LIN {X 0,Y 549.947,Z 550.345,A -85,B 0,C 180,E1 -11066.532,E2 -11066.532} C_VEL
LIN {X 0,Y 549.396,Z 557.599,A -85,B 0,C 180,E1 -11067.808,E2 -11067.808} C_VEL
LIN {X 0,Y 549.182,Z 562.629,A -85,B 0,C 180,E1 -11068.904,E2 -11068.904} C_VEL
LIN {X 0,Y 548.851,Z 567.942,A -85,B 0,C 180,E1 -11070.366,E2 -11070.366} C_VEL
LIN {X 0,Y 548.664,Z 570.891,A -85,B 0,C 180,E1 -11071.463,E2 -11071.463} C_VEL
LIN {X 0,Y 548.707,Z 573.631,A -85,B 0,C 180,E1 -11072.927,E2 -11072.927} C_VEL
LIN {X 0,Y 548.574,Z 575.081,A -85,B 0,C 180,E1 -11074.394,E2 -11074.394} C_VEL
LIN {X 0,Y 548.685,Z 575.22,A -85,B 0,C 180,E1 -11075.862,E2 -11075.862} C_VEL
LIN {X 0,Y 548.777,Z 574.076,A -85,B 0,C 180,E1 -11077.333,E2 -11077.333} C_VEL
LIN {X 0,Y 548.924,Z 571.601,A -85,B 0,C 180,E1 -11078.808,E2 -11078.808} C_VEL
LIN {X 0,Y 549.304,Z 567.682,A -85,B 0,C 180,E1 -11080.284,E2 -11080.284} C_VEL
LIN {X 0,Y 549.668,Z 562.23,A -85,B 0,C 180,E1 -11081.765,E2 -11081.765} C_VEL
LIN {X 0,Y 550.064,Z 557.037,A -85,B 0,C 180,E1 -11082.876,E2 -11082.876} C_VEL
LIN {X 0,Y 550.653,Z 549.525,A -85,B 0,C 180,E1 -11084.174,E2 -11084.174} C_VEL
LIN {X 0,Y 551.216,Z 542.172,A -85,B 0,C 180,E1 -11085.223,E2 -11085.223} C_VEL
LIN {X 0,Y 551.874,Z 532.144,A -85,B 0,C 180,E1 -11086.404,E2 -11086.404} C_VEL
LIN {X 0,Y 552.495,Z 521.544,A -85,B 0,C 180,E1 -11087.429,E2 -11087.429} C_VEL
LIN {X 0,Y 553.106,Z 510.224,A -85,B 0,C 180,E1 -11088.328,E2 -11088.328} C_VEL
LIN {X 0,Y 553.739,Z 498.155,A -85,B 0,C 180,E1 -11089.105,E2 -11089.105} C_VEL
LIN {X 0,Y 554.247,Z 484.443,A -85,B 0,C 180,E1 -11089.807,E2 -11089.807} C_VEL
LIN {X 0,Y 554.553,Z 471.078,A -85,B 0,C 180,E1 -11090.325,E2 -11090.325} C_VEL
LIN {X 0,Y 554.726,Z 456.438,A -85,B 0,C 180,E1 -11090.725,E2 -11090.725} C_VEL
LIN {X 0,Y 554.878,Z 439.3,A -85,B 0,C 180,E1 -11091.001,E2 -11091.001} C_VEL
LIN {X 0,Y 555.689,Z 346.431,A -85,B 0,C 180,E1 -11092.217,E2 -11092.217} C_VEL
LIN {X 0,Y 549.268,Z 330.203,A -85,B 0,C 180,E1 -11092.678,E2 -11092.678} C_VEL
LIN {X 0,Y 549.162,Z 329.646,A -85,B 0,C 180,E1 -11092.721,E2 -11092.721} C_VEL
LIN {X 0,Y 549.175,Z 329.64,A -85,B 0,C 180,E1 -11095.099,E2 -11095.099} C_VEL
LIN {X 0,Y 549.187,Z 329.634,A -85,B 0,C 180,E1 -11098.158,E2 -11098.158} C_VEL
LIN {X 0,Y 549.165,Z 329.637,A -85,B 0,C 180,E1 -11100.677,E2 -11100.677} C_VEL
LIN {X 0,Y 549.119,Z 329.639,A -85,B 0,C 180,E1 -11103.264,E2 -11103.264} C_VEL
LIN {X 0,Y 549.15,Z 329.64,A -85,B 0,C 180,E1 -11105.926,E2 -11105.926} C_VEL
LIN {X 0,Y 549.129,Z 329.638,A -85,B 0,C 180,E1 -11108.914,E2 -11108.914} C_VEL
LIN {X 0,Y 549.137,Z 329.639,A -85,B 0,C 180,E1 -11111.551,E2 -11111.551} C_VEL
LIN {X 0,Y 549.203,Z 329.629,A -85,B 0,C 180,E1 -11114.545,E2 -11114.545} C_VEL
LIN {X 0,Y 549.154,Z 329.636,A -85,B 0,C 180,E1 -11117.467,E2 -11117.467} C_VEL
LIN {X 0,Y 549.137,Z 329.636,A -85,B 0,C 180,E1 -11120.374,E2 -11120.374} C_VEL
LIN {X 0,Y 549.139,Z 329.617,A -85,B 0,C 180,E1 -11123.474,E2 -11123.474} C_VEL
LIN {X 0,Y 549.147,Z 329.637,A -85,B 0,C 180,E1 -11126.005,E2 -11126.005} C_VEL
LIN {X 0,Y 549.161,Z 329.628,A -85,B 0,C 180,E1 -11128.713,E2 -11128.713} C_VEL
LIN {X 0,Y 549.175,Z 329.629,A -85,B 0,C 180,E1 -11131.009,E2 -11131.009} C_VEL
LIN {X 0,Y 549.178,Z 329.634,A -85,B 0,C 180,E1 -11133.486,E2 -11133.486} C_VEL
LIN {X 0,Y 549.163,Z 329.639,A -85,B 0,C 180,E1 -11135.911,E2 -11135.911} C_VEL
LIN {X 0,Y 549.18,Z 329.627,A -85,B 0,C 180,E1 -11139.076,E2 -11139.076} C_VEL
LIN {X 0,Y 549.182,Z 329.642,A -85,B 0,C 180,E1 -11141.406,E2 -11141.406} C_VEL
LIN {X 0,Y 549.194,Z 329.638,A -85,B 0,C 180,E1 -11142.268,E2 -11142.268} C_VEL
LIN {X 0,Y 553.527,Z 343.362,A -85,B 0,C 180,E1 -11142.596,E2 -11142.596} C_VEL
LIN {X 0,Y 552.255,Z 449.713,A -85,B 0,C 180,E1 -11144.222,E2 -11144.222} C_VEL
LIN {X 0,Y 552.112,Z 464.877,A -85,B 0,C 180,E1 -11144.612,E2 -11144.612} C_VEL
LIN {X 0,Y 551.849,Z 479.41,A -85,B 0,C 180,E1 -11145.143,E2 -11145.143} C_VEL
LIN {X 0,Y 551.501,Z 492.173,A -85,B 0,C 180,E1 -11145.754,E2 -11145.754} C_VEL
LIN {X 0,Y 551.121,Z 504.477,A -85,B 0,C 180,E1 -11146.494,E2 -11146.494} C_VEL
LIN {X 0,Y 550.667,Z 516.942,A -85,B 0,C 180,E1 -11147.418,E2 -11147.418} C_VEL
LIN {X 0,Y 550.22,Z 527.741,A -85,B 0,C 180,E1 -11148.39,E2 -11148.39} C_VEL
LIN {X 0,Y 549.971,Z 536.697,A -85,B 0,C 180,E1 -11149.358,E2 -11149.358} C_VEL
LIN {X 0,Y 549.516,Z 545.315,A -85,B 0,C 180,E1 -11150.462,E2 -11150.462} C_VEL
LIN {X 0,Y 549.197,Z 553.545,A -85,B 0,C 180,E1 -11151.75,E2 -11151.75} C_VEL
LIN {X 0,Y 548.936,Z 560.126,A -85,B 0,C 180,E1 -11153.037,E2 -11153.037} C_VEL
LIN {X 0,Y 548.769,Z 564.687,A -85,B 0,C 180,E1 -11154.139,E2 -11154.139} C_VEL
LIN {X 0,Y 548.596,Z 569.27,A -85,B 0,C 180,E1 -11155.606,E2 -11155.606} C_VEL
LIN {X 0,Y 548.655,Z 572.352,A -85,B 0,C 180,E1 -11157.073,E2 -11157.073} C_VEL
LIN {X 0,Y 548.562,Z 574.044,A -85,B 0,C 180,E1 -11158.536,E2 -11158.536} C_VEL
LIN {X 0,Y 548.463,Z 574.349,A -85,B 0,C 180,E1 -11160,E2 -11160} C_VEL
LIN {X 0,Y 548.586,Z 573.208,A -85,B 0,C 180,E1 -11161.463,E2 -11161.463} C_VEL
LIN {X 0,Y 548.967,Z 570.638,A -85,B 0,C 180,E1 -11162.925,E2 -11162.925} C_VEL
LIN {X 0,Y 549.423,Z 566.6,A -85,B 0,C 180,E1 -11164.387,E2 -11164.387} C_VEL
LIN {X 0,Y 549.419,Z 562.553,A -85,B 0,C 180,E1 -11165.487,E2 -11165.487} C_VEL
LIN {X 0,Y 549.926,Z 557.46,A -85,B 0,C 180,E1 -11166.582,E2 -11166.582} C_VEL
LIN {X 0,Y 550.477,Z 550.127,A -85,B 0,C 180,E1 -11167.862,E2 -11167.862} C_VEL
LIN {X 0,Y 550.884,Z 542.443,A -85,B 0,C 180,E1 -11168.961,E2 -11168.961} C_VEL
LIN {X 0,Y 551.383,Z 533.157,A -85,B 0,C 180,E1 -11170.059,E2 -11170.059} C_VEL
LIN {X 0,Y 551.887,Z 522.846,A -85,B 0,C 180,E1 -11171.067,E2 -11171.067} C_VEL
LIN {X 0,Y 552.536,Z 511.383,A -85,B 0,C 180,E1 -11171.981,E2 -11171.981} C_VEL
LIN {X 0,Y 553.175,Z 499.168,A -85,B 0,C 180,E1 -11172.772,E2 -11172.772} C_VEL
LIN {X 0,Y 553.575,Z 486.327,A -85,B 0,C 180,E1 -11173.444,E2 -11173.444} C_VEL
LIN {X 0,Y 553.859,Z 472.723,A -85,B 0,C 180,E1 -11173.997,E2 -11173.997} C_VEL
LIN {X 0,Y 554.047,Z 458.452,A -85,B 0,C 180,E1 -11174.412,E2 -11174.412} C_VEL
LIN {X 0,Y 554.314,Z 436.957,A -85,B 0,C 180,E1 -11174.802,E2 -11174.802} C_VEL
LIN {X 0,Y 556.216,Z 346.413,A -85,B 0,C 180,E1 -11176.312,E2 -11176.312} C_VEL
LIN {X 0,Y 550.079,Z 332.219,A -85,B 0,C 180,E1 -11176.868,E2 -11176.868} C_VEL
LIN {X 0,Y 549.231,Z 329.633,A -85,B 0,C 180,E1 -11176.963,E2 -11176.963} C_VEL
LIN {X 0,Y 549.198,Z 329.636,A -85,B 0,C 180,E1 -11180.142,E2 -11180.142} C_VEL
LIN {X 0,Y 549.204,Z 329.635,A -85,B 0,C 180,E1 -11182.496,E2 -11182.496} C_VEL
LIN {X 0,Y 549.176,Z 329.634,A -85,B 0,C 180,E1 -11185.099,E2 -11185.099} C_VEL
LIN {X 0,Y 549.208,Z 329.633,A -85,B 0,C 180,E1 -11188.157,E2 -11188.157} C_VEL
LIN {X 0,Y 549.179,Z 329.632,A -85,B 0,C 180,E1 -11190.675,E2 -11190.675} C_VEL
LIN {X 0,Y 549.169,Z 329.637,A -85,B 0,C 180,E1 -11193.261,E2 -11193.261} C_VEL
LIN {X 0,Y 549.241,Z 329.624,A -85,B 0,C 180,E1 -11195.919,E2 -11195.919} C_VEL
LIN {X 0,Y 549.156,Z 329.631,A -85,B 0,C 180,E1 -11198.917,E2 -11198.917} C_VEL
LIN {X 0,Y 549.152,Z 329.635,A -85,B 0,C 180,E1 -11201.549,E2 -11201.549} C_VEL
LIN {X 0,Y 549.201,Z 329.626,A -85,B 0,C 180,E1 -11204.544,E2 -11204.544} C_VEL
LIN {X 0,Y 549.151,Z 329.636,A -85,B 0,C 180,E1 -11207.466,E2 -11207.466} C_VEL
LIN {X 0,Y 549.135,Z 329.639,A -85,B 0,C 180,E1 -11210.374,E2 -11210.374} C_VEL
LIN {X 0,Y 549.137,Z 329.639,A -85,B 0,C 180,E1 -11213.474,E2 -11213.474} C_VEL
LIN {X 0,Y 549.134,Z 329.634,A -85,B 0,C 180,E1 -11216.007,E2 -11216.007} C_VEL
LIN {X 0,Y 549.158,Z 329.641,A -85,B 0,C 180,E1 -11218.713,E2 -11218.713} C_VEL
LIN {X 0,Y 549.206,Z 329.796,A -85,B 0,C 180,E1 -11220.566,E2 -11220.566} C_VEL
LIN {X 0,Y 552.802,Z 345.817,A -85,B 0,C 180,E1 -11222.695,E2 -11222.695} C_VEL
LIN {X 0,Y 553.853,Z 352.332,A -85,B 0,C 180,E1 -11223.525,E2 -11223.525} C_VEL
LIN {X 0,Y 552.715,Z 372.997,A -85,B 0,C 180,E1 -11225.943,E2 -11225.943} C_VEL
LIN {X 0,Y 551.503,Z 397.502,A -85,B 0,C 180,E1 -11228.779,E2 -11228.779} C_VEL
LIN {X 0,Y 550.466,Z 420.802,A -85,B 0,C 180,E1 -11231.451,E2 -11231.451} C_VEL
LIN {X 0,Y 550.27,Z 427.795,A -85,B 0,C 180,E1 -11232.252,E2 -11232.252} C_VEL
LIN {X 0,Y 553.911,Z 457.37,A -85,B 0,C 180,E1 -11232.779,E2 -11232.779} C_VEL
LIN {X 0,Y 554.662,Z 468.125,A -85,B 0,C 180,E1 -11232.948,E2 -11232.948} C_VEL
LIN {X 0,Y 553.636,Z 567.72,A -85,B 0,C 180,E1 -11234.261,E2 -11234.261} C_VEL
LIN {X 0,Y 553.075,Z 582.303,A -85,B 0,C 180,E1 -11234.6,E2 -11234.6} C_VEL
LIN {X 0,Y 552.321,Z 596.222,A -85,B 0,C 180,E1 -11235.072,E2 -11235.072} C_VEL
LIN {X 0,Y 551.604,Z 609.218,A -85,B 0,C 180,E1 -11235.663,E2 -11235.663} C_VEL
LIN {X 0,Y 550.874,Z 621.854,A -85,B 0,C 180,E1 -11236.395,E2 -11236.395} C_VEL
LIN {X 0,Y 549.969,Z 637.761,A -85,B 0,C 180,E1 -11237.496,E2 -11237.496} C_VEL
LIN {X 0,Y 549.523,Z 649.094,A -85,B 0,C 180,E1 -11238.325,E2 -11238.325} C_VEL
LIN {X 0,Y 549.089,Z 660.252,A -85,B 0,C 180,E1 -11239.321,E2 -11239.321} C_VEL
LIN {X 0,Y 548.678,Z 670.589,A -85,B 0,C 180,E1 -11240.447,E2 -11240.447} C_VEL
LIN {X 0,Y 548.335,Z 678.978,A -85,B 0,C 180,E1 -11241.552,E2 -11241.552} C_VEL
LIN {X 0,Y 548.111,Z 686.974,A -85,B 0,C 180,E1 -11242.842,E2 -11242.842} C_VEL
LIN {X 0,Y 547.996,Z 693.354,A -85,B 0,C 180,E1 -11244.131,E2 -11244.131} C_VEL
LIN {X 0,Y 547.888,Z 697.67,A -85,B 0,C 180,E1 -11245.233,E2 -11245.233} C_VEL
LIN {X 0,Y 547.844,Z 701.065,A -85,B 0,C 180,E1 -11246.335,E2 -11246.335} C_VEL
LIN {X 0,Y 547.83,Z 704.197,A -85,B 0,C 180,E1 -11247.802,E2 -11247.802} C_VEL
LIN {X 0,Y 547.771,Z 705.866,A -85,B 0,C 180,E1 -11249.267,E2 -11249.267} C_VEL
LIN {X 0,Y 547.77,Z 706.099,A -85,B 0,C 180,E1 -11250.733,E2 -11250.733} C_VEL
LIN {X 0,Y 547.832,Z 704.902,A -85,B 0,C 180,E1 -11252.198,E2 -11252.198} C_VEL
LIN {X 0,Y 547.856,Z 702.24,A -85,B 0,C 180,E1 -11253.665,E2 -11253.665} C_VEL
LIN {X 0,Y 547.919,Z 699.228,A -85,B 0,C 180,E1 -11254.766,E2 -11254.766} C_VEL
LIN {X 0,Y 548.047,Z 695.312,A -85,B 0,C 180,E1 -11255.868,E2 -11255.868} C_VEL
LIN {X 0,Y 548.21,Z 690.434,A -85,B 0,C 180,E1 -11256.972,E2 -11256.972} C_VEL
LIN {X 0,Y 548.487,Z 683.347,A -85,B 0,C 180,E1 -11258.26,E2 -11258.26} C_VEL
LIN {X 0,Y 548.849,Z 675.914,A -85,B 0,C 180,E1 -11259.365,E2 -11259.365} C_VEL
LIN {X 0,Y 549.334,Z 665.904,A -85,B 0,C 180,E1 -11260.586,E2 -11260.586} C_VEL
LIN {X 0,Y 549.866,Z 655.087,A -85,B 0,C 180,E1 -11261.667,E2 -11261.667} C_VEL
LIN {X 0,Y 550.482,Z 643.898,A -85,B 0,C 180,E1 -11262.586,E2 -11262.586} C_VEL
LIN {X 0,Y 551.09,Z 631.56,A -85,B 0,C 180,E1 -11263.412,E2 -11263.412} C_VEL
LIN {X 0,Y 551.731,Z 617.816,A -85,B 0,C 180,E1 -11264.146,E2 -11264.146} C_VEL
LIN {X 0,Y 552.216,Z 604.549,A -85,B 0,C 180,E1 -11264.696,E2 -11264.696} C_VEL
LIN {X 0,Y 552.728,Z 589.51,A -85,B 0,C 180,E1 -11265.151,E2 -11265.151} C_VEL
LIN {X 0,Y 553.143,Z 572.743,A -85,B 0,C 180,E1 -11265.47,E2 -11265.47} C_VEL
LIN {X 0,Y 555.059,Z 479.753,A -85,B 0,C 180,E1 -11267.027,E2 -11267.027} C_VEL
LIN {X 0,Y 555.244,Z 464.014,A -85,B 0,C 180,E1 -11267.31,E2 -11267.31} C_VEL
LIN {X 0,Y 553.176,Z 441.384,A -85,B 0,C 180,E1 -11267.832,E2 -11267.832} C_VEL
LIN {X 0,Y 552.115,Z 432.409,A -85,B 0,C 180,E1 -11268.089,E2 -11268.089} C_VEL
LIN {X 0,Y 550.207,Z 415.419,A -85,B 0,C 180,E1 -11268.75,E2 -11268.75} C_VEL
LIN {X 0,Y 551.164,Z 391.674,A -85,B 0,C 180,E1 -11271.43,E2 -11271.43} C_VEL
LIN {X 0,Y 552.137,Z 367.93,A -85,B 0,C 180,E1 -11274.13,E2 -11274.13} C_VEL
LIN {X 0,Y 552.954,Z 348.856,A -85,B 0,C 180,E1 -11276.318,E2 -11276.318} C_VEL
LIN {X 0,Y 549.905,Z 332.981,A -85,B 0,C 180,E1 -11278.3,E2 -11278.3} C_VEL
LIN {X 0,Y 549.19,Z 329.635,A -85,B 0,C 180,E1 -11278.746,E2 -11278.746} C_VEL
LIN {X 0,Y 549.151,Z 329.642,A -85,B 0,C 180,E1 -11281.531,E2 -11281.531} C_VEL
LIN {X 0,Y 549.129,Z 329.638,A -85,B 0,C 180,E1 -11284.142,E2 -11284.142} C_VEL
LIN {X 0,Y 549.116,Z 329.642,A -85,B 0,C 180,E1 -11286.836,E2 -11286.836} C_VEL
LIN {X 0,Y 549.154,Z 329.636,A -85,B 0,C 180,E1 -11290.067,E2 -11290.067} C_VEL
LIN {X 0,Y 549.11,Z 329.643,A -85,B 0,C 180,E1 -11292.537,E2 -11292.537} C_VEL
LIN {X 0,Y 549.198,Z 329.634,A -85,B 0,C 180,E1 -11295.455,E2 -11295.455} C_VEL
LIN {X 0,Y 549.148,Z 329.638,A -85,B 0,C 180,E1 -11298.812,E2 -11298.812} C_VEL
LIN {X 0,Y 549.128,Z 329.642,A -85,B 0,C 180,E1 -11301.316,E2 -11301.316} C_VEL
LIN {X 0,Y 549.193,Z 329.634,A -85,B 0,C 180,E1 -11304.078,E2 -11304.078} C_VEL
LIN {X 0,Y 549.131,Z 329.646,A -85,B 0,C 180,E1 -11306.737,E2 -11306.737} C_VEL
LIN {X 0,Y 549.198,Z 329.821,A -85,B 0,C 180,E1 -11309.591,E2 -11309.591} C_VEL
LIN {X 0,Y 553.46,Z 343.452,A -85,B 0,C 180,E1 -11311.461,E2 -11311.461} C_VEL
LIN {X 0,Y 555.988,Z 354.319,A -85,B 0,C 180,E1 -11312.847,E2 -11312.847} C_VEL
LIN {X 0,Y 556.314,Z 357.522,A -85,B 0,C 180,E1 -11313.221,E2 -11313.221} C_VEL
LIN {X 0,Y 555.107,Z 383.215,A -85,B 0,C 180,E1 -11315.988,E2 -11315.988} C_VEL
LIN {X 0,Y 553.946,Z 408.488,A -85,B 0,C 180,E1 -11318.683,E2 -11318.683} C_VEL
LIN {X 0,Y 552.882,Z 435.159,A -85,B 0,C 180,E1 -11321.535,E2 -11321.535} C_VEL
LIN {X 0,Y 552.785,Z 440.026,A -85,B 0,C 180,E1 -11322.028,E2 -11322.028} C_VEL
LIN {X 0,Y 555.641,Z 458.614,A -85,B 0,C 180,E1 -11322.508,E2 -11322.508} C_VEL
LIN {X 0,Y 555.992,Z 463.553,A -85,B 0,C 180,E1 -11322.614,E2 -11322.614} C_VEL
LIN {X 0,Y 554.091,Z 550.209,A -85,B 0,C 180,E1 -11324.065,E2 -11324.065} C_VEL
LIN {X 0,Y 553.386,Z 581.221,A -85,B 0,C 180,E1 -11324.585,E2 -11324.585} C_VEL
LIN {X 0,Y 552.951,Z 594.971,A -85,B 0,C 180,E1 -11324.949,E2 -11324.949} C_VEL
LIN {X 0,Y 552.363,Z 609.631,A -85,B 0,C 180,E1 -11325.496,E2 -11325.496} C_VEL
LIN {X 0,Y 551.764,Z 622.746,A -85,B 0,C 180,E1 -11326.137,E2 -11326.137} C_VEL
LIN {X 0,Y 551.018,Z 636.153,A -85,B 0,C 180,E1 -11326.96,E2 -11326.96} C_VEL
LIN {X 0,Y 550.346,Z 648.168,A -85,B 0,C 180,E1 -11327.878,E2 -11327.878} C_VEL
LIN {X 0,Y 549.67,Z 659.904,A -85,B 0,C 180,E1 -11328.981,E2 -11328.981} C_VEL
LIN {X 0,Y 549.233,Z 669.573,A -85,B 0,C 180,E1 -11330.086,E2 -11330.086} C_VEL
LIN {X 0,Y 548.692,Z 677.61,A -85,B 0,C 180,E1 -11331.188,E2 -11331.188} C_VEL
LIN {X 0,Y 548.413,Z 684.289,A -85,B 0,C 180,E1 -11332.293,E2 -11332.293} C_VEL
LIN {X 0,Y 548.172,Z 689.823,A -85,B 0,C 180,E1 -11333.397,E2 -11333.397} C_VEL
LIN {X 0,Y 547.907,Z 695.618,A -85,B 0,C 180,E1 -11334.866,E2 -11334.866} C_VEL
LIN {X 0,Y 547.872,Z 698.27,A -85,B 0,C 180,E1 -11335.726,E2 -11335.726} C_VEL
LIN {X 0,Y 547.8,Z 701.322,A -85,B 0,C 180,E1 -11337.068,E2 -11337.068} C_VEL
LIN {X 0,Y 547.724,Z 703.252,A -85,B 0,C 180,E1 -11338.535,E2 -11338.535} C_VEL
LIN {X 0,Y 547.712,Z 703.757,A -85,B 0,C 180,E1 -11340,E2 -11340} C_VEL
LIN {X 0,Y 547.723,Z 702.852,A -85,B 0,C 180,E1 -11341.466,E2 -11341.466} C_VEL
LIN {X 0,Y 547.796,Z 700.526,A -85,B 0,C 180,E1 -11342.932,E2 -11342.932} C_VEL
LIN {X 0,Y 547.822,Z 696.729,A -85,B 0,C 180,E1 -11344.4,E2 -11344.4} C_VEL
LIN {X 0,Y 547.913,Z 692.805,A -85,B 0,C 180,E1 -11345.502,E2 -11345.502} C_VEL
LIN {X 0,Y 548.026,Z 687.924,A -85,B 0,C 180,E1 -11346.606,E2 -11346.606} C_VEL
LIN {X 0,Y 548.296,Z 680.845,A -85,B 0,C 180,E1 -11347.894,E2 -11347.894} C_VEL
LIN {X 0,Y 548.634,Z 672.058,A -85,B 0,C 180,E1 -11349.183,E2 -11349.183} C_VEL
LIN {X 0,Y 549.083,Z 662.859,A -85,B 0,C 180,E1 -11350.288,E2 -11350.288} C_VEL
LIN {X 0,Y 549.521,Z 651.636,A -85,B 0,C 180,E1 -11351.395,E2 -11351.395} C_VEL
LIN {X 0,Y 550.03,Z 640.249,A -85,B 0,C 180,E1 -11352.316,E2 -11352.316} C_VEL
LIN {X 0,Y 550.577,Z 627.739,A -85,B 0,C 180,E1 -11353.145,E2 -11353.145} C_VEL
LIN {X 0,Y 551.131,Z 613.829,A -85,B 0,C 180,E1 -11353.88,E2 -11353.88} C_VEL
LIN {X 0,Y 551.589,Z 600.184,A -85,B 0,C 180,E1 -11354.431,E2 -11354.431} C_VEL
LIN {X 0,Y 551.934,Z 585.273,A -85,B 0,C 180,E1 -11354.868,E2 -11354.868} C_VEL
LIN {X 0,Y 552.26,Z 569.363,A -85,B 0,C 180,E1 -11355.165,E2 -11355.165} C_VEL
LIN {X 0,Y 553.706,Z 459.872,A -85,B 0,C 180,E1 -11356.838,E2 -11356.838} C_VEL
LIN {X 0,Y 551.279,Z 439.437,A -85,B 0,C 180,E1 -11357.241,E2 -11357.241} C_VEL
LIN {X 0,Y 552.337,Z 407.939,A -85,B 0,C 180,E1 -11360.61,E2 -11360.61} C_VEL
LIN {X 0,Y 553.42,Z 379.174,A -85,B 0,C 180,E1 -11363.694,E2 -11363.694} C_VEL
LIN {X 0,Y 554.364,Z 353.607,A -85,B 0,C 180,E1 -11366.448,E2 -11366.448} C_VEL
LIN {X 0,Y 553.32,Z 347.877,A -85,B 0,C 180,E1 -11367.112,E2 -11367.112} C_VEL
LIN {X 0,Y 549.207,Z 329.634,A -85,B 0,C 180,E1 -11369.303,E2 -11369.303} C_VEL
LIN {X 0,Y 549.16,Z 329.633,A -85,B 0,C 180,E1 -11372.392,E2 -11372.392} C_VEL
LIN {X 0,Y 549.233,Z 329.632,A -85,B 0,C 180,E1 -11375.294,E2 -11375.294} C_VEL
LIN {X 0,Y 549.17,Z 329.633,A -85,B 0,C 180,E1 -11377.751,E2 -11377.751} C_VEL
LIN {X 0,Y 549.177,Z 329.632,A -85,B 0,C 180,E1 -11380.578,E2 -11380.578} C_VEL
LIN {X 0,Y 549.187,Z 329.631,A -85,B 0,C 180,E1 -11383.53,E2 -11383.53} C_VEL
LIN {X 0,Y 549.187,Z 329.632,A -85,B 0,C 180,E1 -11386.471,E2 -11386.471} C_VEL
LIN {X 0,Y 549.187,Z 329.63,A -85,B 0,C 180,E1 -11389.423,E2 -11389.423} C_VEL
LIN {X 0,Y 549.171,Z 329.634,A -85,B 0,C 180,E1 -11392.259,E2 -11392.259} C_VEL
LIN {X 0,Y 549.22,Z 329.629,A -85,B 0,C 180,E1 -11394.977,E2 -11394.977} C_VEL
LIN {X 0,Y 549.159,Z 329.633,A -85,B 0,C 180,E1 -11397.608,E2 -11397.608} C_VEL
LIN {X 0,Y 549.193,Z 329.633,A -85,B 0,C 180,E1 -11400.171,E2 -11400.171} C_VEL
LIN {X 0,Y 549.197,Z 329.632,A -85,B 0,C 180,E1 -11402.668,E2 -11402.668} C_VEL
LIN {X 0,Y 549.175,Z 329.634,A -85,B 0,C 180,E1 -11405.912,E2 -11405.912} C_VEL
LIN {X 0,Y 549.213,Z 329.629,A -85,B 0,C 180,E1 -11408.594,E2 -11408.594} C_VEL
LIN {X 0,Y 549.204,Z 329.628,A -85,B 0,C 180,E1 -11410.778,E2 -11410.778} C_VEL
LIN {X 0,Y 548.513,Z 329.715,A -85,B 0,C 180,E1 -11411.391,E2 -11411.391} C_VEL
LIN {X 0,Y 545.65,Z 330.074,A -85,B 0,C 180,E1 -11412.385,E2 -11412.385} C_VEL
LIN {X 0,Y 543.251,Z 330.371,A -85,B 0,C 180,E1 -11413.186,E2 -11413.186} C_VEL
LIN {X 0,Y 542.234,Z 330.501,A -85,B 0,C 180,E1 -11413.804,E2 -11413.804} C_VEL
LIN {X 0,Y 542.157,Z 330.507,A -85,B 0,C 180,E1 -11414.013,E2 -11414.013} C_VEL
LIN {X 0,Y 542.187,Z 330.503,A -85,B 0,C 180,E1 -11416.553,E2 -11416.553} C_VEL
LIN {X 0,Y 542.204,Z 330.512,A -85,B 0,C 180,E1 -11417.806,E2 -11417.806} C_VEL
LIN {X 0,Y 547.413,Z 345.743,A -85,B 0,C 180,E1 -11418.169,E2 -11418.169} C_VEL
LIN {X 0,Y 546.695,Z 448.46,A -85,B 0,C 180,E1 -11419.527,E2 -11419.527} C_VEL
LIN {X 0,Y 546.584,Z 462.819,A -85,B 0,C 180,E1 -11419.828,E2 -11419.828} C_VEL
LIN {X 0,Y 546.324,Z 476.603,A -85,B 0,C 180,E1 -11420.266,E2 -11420.266} C_VEL
LIN {X 0,Y 545.924,Z 490.402,A -85,B 0,C 180,E1 -11420.864,E2 -11420.864} C_VEL
LIN {X 0,Y 545.501,Z 502.571,A -85,B 0,C 180,E1 -11421.547,E2 -11421.547} C_VEL
LIN {X 0,Y 545.032,Z 515.126,A -85,B 0,C 180,E1 -11422.431,E2 -11422.431} C_VEL
LIN {X 0,Y 544.42,Z 525.858,A -85,B 0,C 180,E1 -11423.351,E2 -11423.351} C_VEL
LIN {X 0,Y 543.85,Z 534.859,A -85,B 0,C 180,E1 -11424.272,E2 -11424.272} C_VEL
LIN {X 0,Y 543.301,Z 543.874,A -85,B 0,C 180,E1 -11425.378,E2 -11425.378} C_VEL
LIN {X 0,Y 542.839,Z 552.475,A -85,B 0,C 180,E1 -11426.671,E2 -11426.671} C_VEL
LIN {X 0,Y 542.364,Z 558.575,A -85,B 0,C 180,E1 -11427.78,E2 -11427.78} C_VEL
LIN {X 0,Y 541.988,Z 565.029,A -85,B 0,C 180,E1 -11429.26,E2 -11429.26} C_VEL
LIN {X 0,Y 541.672,Z 569.89,A -85,B 0,C 180,E1 -11430.741,E2 -11430.741} C_VEL
LIN {X 0,Y 541.676,Z 573.274,A -85,B 0,C 180,E1 -11432.223,E2 -11432.223} C_VEL
LIN {X 0,Y 541.642,Z 575.325,A -85,B 0,C 180,E1 -11433.707,E2 -11433.707} C_VEL
LIN {X 0,Y 541.602,Z 576.095,A -85,B 0,C 180,E1 -11435.232,E2 -11435.232} C_VEL
LIN {X 0,Y 541.683,Z 575.551,A -85,B 0,C 180,E1 -11436.683,E2 -11436.683} C_VEL
LIN {X 0,Y 541.825,Z 573.703,A -85,B 0,C 180,E1 -11438.175,E2 -11438.175} C_VEL
LIN {X 0,Y 542.075,Z 570.474,A -85,B 0,C 180,E1 -11439.671,E2 -11439.671} C_VEL
LIN {X 0,Y 542.472,Z 565.763,A -85,B 0,C 180,E1 -11441.168,E2 -11441.168} C_VEL
LIN {X 0,Y 542.979,Z 559.429,A -85,B 0,C 180,E1 -11442.668,E2 -11442.668} C_VEL
LIN {X 0,Y 543.561,Z 552.345,A -85,B 0,C 180,E1 -11443.982,E2 -11443.982} C_VEL
LIN {X 0,Y 544.248,Z 543.821,A -85,B 0,C 180,E1 -11445.26,E2 -11445.26} C_VEL
LIN {X 0,Y 544.919,Z 534.265,A -85,B 0,C 180,E1 -11446.427,E2 -11446.427} C_VEL
LIN {X 0,Y 545.571,Z 523.941,A -85,B 0,C 180,E1 -11447.464,E2 -11447.464} C_VEL
LIN {X 0,Y 546.204,Z 512.848,A -85,B 0,C 180,E1 -11448.383,E2 -11448.383} C_VEL
LIN {X 0,Y 546.865,Z 501.344,A -85,B 0,C 180,E1 -11449.161,E2 -11449.161} C_VEL
LIN {X 0,Y 547.383,Z 489.261,A -85,B 0,C 180,E1 -11449.822,E2 -11449.822} C_VEL
LIN {X 0,Y 547.673,Z 477.204,A -85,B 0,C 180,E1 -11450.348,E2 -11450.348} C_VEL
LIN {X 0,Y 547.954,Z 463.069,A -85,B 0,C 180,E1 -11450.801,E2 -11450.801} C_VEL
LIN {X 0,Y 548.087,Z 449.512,A -85,B 0,C 180,E1 -11451.091,E2 -11451.091} C_VEL
LIN {X 0,Y 548.973,Z 348.102,A -85,B 0,C 180,E1 -11452.445,E2 -11452.445} C_VEL
LIN {X 0,Y 542.196,Z 330.857,A -85,B 0,C 180,E1 -11452.943,E2 -11452.943} C_VEL
LIN {X 0,Y 542.135,Z 330.521,A -85,B 0,C 180,E1 -11452.957,E2 -11452.957} C_VEL
LIN {X 0,Y 542.127,Z 330.517,A -85,B 0,C 180,E1 -11455.254,E2 -11455.254} C_VEL
LIN {X 0,Y 542.135,Z 330.514,A -85,B 0,C 180,E1 -11457.718,E2 -11457.718} C_VEL
LIN {X 0,Y 542.125,Z 330.516,A -85,B 0,C 180,E1 -11460.258,E2 -11460.258} C_VEL
LIN {X 0,Y 542.09,Z 330.516,A -85,B 0,C 180,E1 -11462.872,E2 -11462.872} C_VEL
LIN {X 0,Y 542.11,Z 330.513,A -85,B 0,C 180,E1 -11465.552,E2 -11465.552} C_VEL
LIN {X 0,Y 542.085,Z 330.523,A -85,B 0,C 180,E1 -11468.333,E2 -11468.333} C_VEL
LIN {X 0,Y 542.105,Z 330.514,A -85,B 0,C 180,E1 -11471.221,E2 -11471.221} C_VEL
LIN {X 0,Y 542.153,Z 330.505,A -85,B 0,C 180,E1 -11474.717,E2 -11474.717} C_VEL
LIN {X 0,Y 542.108,Z 330.513,A -85,B 0,C 180,E1 -11477.433,E2 -11477.433} C_VEL
LIN {X 0,Y 542.121,Z 330.515,A -85,B 0,C 180,E1 -11479.757,E2 -11479.757} C_VEL
LIN {X 0,Y 542.088,Z 330.495,A -85,B 0,C 180,E1 -11482.605,E2 -11482.605} C_VEL
LIN {X 0,Y 542.115,Z 330.502,A -85,B 0,C 180,E1 -11485.354,E2 -11485.354} C_VEL
LIN {X 0,Y 542.112,Z 330.512,A -85,B 0,C 180,E1 -11488.011,E2 -11488.011} C_VEL
LIN {X 0,Y 542.152,Z 330.504,A -85,B 0,C 180,E1 -11490.597,E2 -11490.597} C_VEL
LIN {X 0,Y 542.121,Z 330.508,A -85,B 0,C 180,E1 -11493.114,E2 -11493.114} C_VEL
LIN {X 0,Y 542.134,Z 330.51,A -85,B 0,C 180,E1 -11495.578,E2 -11495.578} C_VEL
LIN {X 0,Y 542.145,Z 330.502,A -85,B 0,C 180,E1 -11498.792,E2 -11498.792} C_VEL
LIN {X 0,Y 542.152,Z 330.513,A -85,B 0,C 180,E1 -11501.156,E2 -11501.156} C_VEL
LIN {X 0,Y 542.153,Z 330.516,A -85,B 0,C 180,E1 -11502.099,E2 -11502.099} C_VEL
LIN {X 0,Y 546.645,Z 345.441,A -85,B 0,C 180,E1 -11502.461,E2 -11502.461} C_VEL
LIN {X 0,Y 545.275,Z 451.134,A -85,B 0,C 180,E1 -11504.111,E2 -11504.111} C_VEL
LIN {X 0,Y 545.134,Z 466.248,A -85,B 0,C 180,E1 -11504.511,E2 -11504.511} C_VEL
LIN {X 0,Y 544.875,Z 480.284,A -85,B 0,C 180,E1 -11505.035,E2 -11505.035} C_VEL
LIN {X 0,Y 544.506,Z 493.145,A -85,B 0,C 180,E1 -11505.662,E2 -11505.662} C_VEL
LIN {X 0,Y 544.111,Z 505.413,A -85,B 0,C 180,E1 -11506.412,E2 -11506.412} C_VEL
LIN {X 0,Y 543.651,Z 517.861,A -85,B 0,C 180,E1 -11507.348,E2 -11507.348} C_VEL
LIN {X 0,Y 543.216,Z 527.916,A -85,B 0,C 180,E1 -11508.26,E2 -11508.26} C_VEL
LIN {X 0,Y 542.905,Z 538.394,A -85,B 0,C 180,E1 -11509.406,E2 -11509.406} C_VEL
LIN {X 0,Y 542.456,Z 546.86,A -85,B 0,C 180,E1 -11510.524,E2 -11510.524} C_VEL
LIN {X 0,Y 542.141,Z 554.921,A -85,B 0,C 180,E1 -11511.829,E2 -11511.829} C_VEL
LIN {X 0,Y 541.897,Z 560.582,A -85,B 0,C 180,E1 -11512.946,E2 -11512.946} C_VEL
LIN {X 0,Y 541.678,Z 566.504,A -85,B 0,C 180,E1 -11514.435,E2 -11514.435} C_VEL
LIN {X 0,Y 541.546,Z 569.887,A -85,B 0,C 180,E1 -11515.549,E2 -11515.549} C_VEL
LIN {X 0,Y 541.614,Z 573.04,A -85,B 0,C 180,E1 -11517.035,E2 -11517.035} C_VEL
LIN {X 0,Y 541.516,Z 574.805,A -85,B 0,C 180,E1 -11518.517,E2 -11518.517} C_VEL
LIN {X 0,Y 541.431,Z 575.189,A -85,B 0,C 180,E1 -11520,E2 -11520} C_VEL
LIN {X 0,Y 541.559,Z 574.121,A -85,B 0,C 180,E1 -11521.482,E2 -11521.482} C_VEL
LIN {X 0,Y 541.954,Z 571.605,A -85,B 0,C 180,E1 -11522.963,E2 -11522.963} C_VEL
LIN {X 0,Y 542.425,Z 567.629,A -85,B 0,C 180,E1 -11524.444,E2 -11524.444} C_VEL
LIN {X 0,Y 542.457,Z 563.643,A -85,B 0,C 180,E1 -11525.557,E2 -11525.557} C_VEL
LIN {X 0,Y 542.968,Z 558.614,A -85,B 0,C 180,E1 -11526.667,E2 -11526.667} C_VEL
LIN {X 0,Y 543.551,Z 551.331,A -85,B 0,C 180,E1 -11527.963,E2 -11527.963} C_VEL
LIN {X 0,Y 543.986,Z 543.715,A -85,B 0,C 180,E1 -11529.075,E2 -11529.075} C_VEL
LIN {X 0,Y 544.525,Z 534.522,A -85,B 0,C 180,E1 -11530.187,E2 -11530.187} C_VEL
LIN {X 0,Y 545.066,Z 524.333,A -85,B 0,C 180,E1 -11531.208,E2 -11531.208} C_VEL
LIN {X 0,Y 545.733,Z 513.018,A -85,B 0,C 180,E1 -11532.132,E2 -11532.132} C_VEL
LIN {X 0,Y 546.424,Z 500.356,A -85,B 0,C 180,E1 -11532.969,E2 -11532.969} C_VEL
LIN {X 0,Y 546.859,Z 488.371,A -85,B 0,C 180,E1 -11533.612,E2 -11533.612} C_VEL
LIN {X 0,Y 547.135,Z 475.179,A -85,B 0,C 180,E1 -11534.172,E2 -11534.172} C_VEL
LIN {X 0,Y 547.387,Z 460.911,A -85,B 0,C 180,E1 -11534.615,E2 -11534.615} C_VEL
LIN {X 0,Y 547.634,Z 444.338,A -85,B 0,C 180,E1 -11534.94,E2 -11534.94} C_VEL
LIN {X 0,Y 549.319,Z 363.667,A -85,B 0,C 180,E1 -11536.309,E2 -11536.309} C_VEL
LIN {X 0,Y 549.657,Z 348.15,A -85,B 0,C 180,E1 -11536.585,E2 -11536.585} C_VEL
LIN {X 0,Y 543.222,Z 333.38,A -85,B 0,C 180,E1 -11537.197,E2 -11537.197} C_VEL
LIN {X 0,Y 542.193,Z 330.509,A -85,B 0,C 180,E1 -11537.309,E2 -11537.309} C_VEL
LIN {X 0,Y 542.165,Z 330.511,A -85,B 0,C 180,E1 -11540.415,E2 -11540.415} C_VEL
LIN {X 0,Y 542.143,Z 330.515,A -85,B 0,C 180,E1 -11543.463,E2 -11543.463} C_VEL
LIN {X 0,Y 542.112,Z 330.518,A -85,B 0,C 180,E1 -11546.059,E2 -11546.059} C_VEL
LIN {X 0,Y 542.152,Z 330.508,A -85,B 0,C 180,E1 -11548.557,E2 -11548.557} C_VEL
LIN {X 0,Y 542.125,Z 330.516,A -85,B 0,C 180,E1 -11551.488,E2 -11551.488} C_VEL
LIN {X 0,Y 542.162,Z 330.504,A -85,B 0,C 180,E1 -11554.643,E2 -11554.643} C_VEL
LIN {X 0,Y 542.138,Z 330.508,A -85,B 0,C 180,E1 -11557.39,E2 -11557.39} C_VEL
LIN {X 0,Y 542.106,Z 330.507,A -85,B 0,C 180,E1 -11560.33,E2 -11560.33} C_VEL
LIN {X 0,Y 542.125,Z 330.514,A -85,B 0,C 180,E1 -11563.218,E2 -11563.218} C_VEL
LIN {X 0,Y 542.154,Z 330.505,A -85,B 0,C 180,E1 -11565.76,E2 -11565.76} C_VEL
LIN {X 0,Y 542.109,Z 330.517,A -85,B 0,C 180,E1 -11568.779,E2 -11568.779} C_VEL
LIN {X 0,Y 542.082,Z 330.516,A -85,B 0,C 180,E1 -11571.667,E2 -11571.667} C_VEL
LIN {X 0,Y 542.103,Z 330.518,A -85,B 0,C 180,E1 -11574.49,E2 -11574.49} C_VEL
LIN {X 0,Y 542.099,Z 330.517,A -85,B 0,C 180,E1 -11577.133,E2 -11577.133} C_VEL
LIN {X 0,Y 542.162,Z 330.599,A -85,B 0,C 180,E1 -11580.321,E2 -11580.321} C_VEL
LIN {X 0,Y 545.753,Z 346.591,A -85,B 0,C 180,E1 -11582.481,E2 -11582.481} C_VEL
LIN {X 0,Y 546.974,Z 353.444,A -85,B 0,C 180,E1 -11583.371,E2 -11583.371} C_VEL
LIN {X 0,Y 545.852,Z 373.539,A -85,B 0,C 180,E1 -11585.755,E2 -11585.755} C_VEL
LIN {X 0,Y 544.476,Z 400.252,A -85,B 0,C 180,E1 -11588.887,E2 -11588.887} C_VEL
LIN {X 0,Y 543.307,Z 427.002,A -85,B 0,C 180,E1 -11591.994,E2 -11591.994} C_VEL
LIN {X 0,Y 547.201,Z 458.285,A -85,B 0,C 180,E1 -11592.561,E2 -11592.561} C_VEL
LIN {X 0,Y 547.93,Z 468.395,A -85,B 0,C 180,E1 -11592.723,E2 -11592.723} C_VEL
LIN {X 0,Y 546.869,Z 566.67,A -85,B 0,C 180,E1 -11594.033,E2 -11594.033} C_VEL
LIN {X 0,Y 546.278,Z 581.477,A -85,B 0,C 180,E1 -11594.379,E2 -11594.379} C_VEL
LIN {X 0,Y 545.468,Z 595.972,A -85,B 0,C 180,E1 -11594.88,E2 -11594.88} C_VEL
LIN {X 0,Y 544.711,Z 608.852,A -85,B 0,C 180,E1 -11595.478,E2 -11595.478} C_VEL
LIN {X 0,Y 543.935,Z 621.406,A -85,B 0,C 180,E1 -11596.218,E2 -11596.218} C_VEL
LIN {X 0,Y 543.098,Z 632.871,A -85,B 0,C 180,E1 -11597.051,E2 -11597.051} C_VEL
LIN {X 0,Y 542.475,Z 648.281,A -85,B 0,C 180,E1 -11598.172,E2 -11598.172} C_VEL
LIN {X 0,Y 542.071,Z 659.632,A -85,B 0,C 180,E1 -11599.181,E2 -11599.181} C_VEL
LIN {X 0,Y 541.606,Z 670.081,A -85,B 0,C 180,E1 -11600.321,E2 -11600.321} C_VEL
LIN {X 0,Y 541.272,Z 678.564,A -85,B 0,C 180,E1 -11601.441,E2 -11601.441} C_VEL
LIN {X 0,Y 541.029,Z 686.64,A -85,B 0,C 180,E1 -11602.748,E2 -11602.748} C_VEL
LIN {X 0,Y 540.911,Z 693.089,A -85,B 0,C 180,E1 -11604.054,E2 -11604.054} C_VEL
LIN {X 0,Y 540.804,Z 697.468,A -85,B 0,C 180,E1 -11605.171,E2 -11605.171} C_VEL
LIN {X 0,Y 540.756,Z 700.919,A -85,B 0,C 180,E1 -11606.286,E2 -11606.286} C_VEL
LIN {X 0,Y 540.758,Z 704.102,A -85,B 0,C 180,E1 -11607.773,E2 -11607.773} C_VEL
LIN {X 0,Y 540.687,Z 705.816,A -85,B 0,C 180,E1 -11609.258,E2 -11609.258} C_VEL
LIN {X 0,Y 540.686,Z 706.093,A -85,B 0,C 180,E1 -11610.742,E2 -11610.742} C_VEL
LIN {X 0,Y 540.76,Z 704.933,A -85,B 0,C 180,E1 -11612.227,E2 -11612.227} C_VEL
LIN {X 0,Y 540.77,Z 702.316,A -85,B 0,C 180,E1 -11613.713,E2 -11613.713} C_VEL
LIN {X 0,Y 540.87,Z 698.143,A -85,B 0,C 180,E1 -11615.201,E2 -11615.201} C_VEL
LIN {X 0,Y 541.022,Z 693.974,A -85,B 0,C 180,E1 -11616.318,E2 -11616.318} C_VEL
LIN {X 0,Y 541.196,Z 688.753,A -85,B 0,C 180,E1 -11617.436,E2 -11617.436} C_VEL
LIN {X 0,Y 541.514,Z 681.268,A -85,B 0,C 180,E1 -11618.742,E2 -11618.742} C_VEL
LIN {X 0,Y 542.063,Z 671.919,A -85,B 0,C 180,E1 -11620.046,E2 -11620.046} C_VEL
LIN {X 0,Y 542.56,Z 662.131,A -85,B 0,C 180,E1 -11621.166,E2 -11621.166} C_VEL
LIN {X 0,Y 543.207,Z 651.26,A -85,B 0,C 180,E1 -11622.19,E2 -11622.19} C_VEL
LIN {X 0,Y 543.807,Z 639.25,A -85,B 0,C 180,E1 -11623.121,E2 -11623.121} C_VEL
LIN {X 0,Y 544.569,Z 625.825,A -85,B 0,C 180,E1 -11623.956,E2 -11623.956} C_VEL
LIN {X 0,Y 545.112,Z 612.594,A -85,B 0,C 180,E1 -11624.606,E2 -11624.606} C_VEL
LIN {X 0,Y 545.697,Z 598.348,A -85,B 0,C 180,E1 -11625.137,E2 -11625.137} C_VEL
LIN {X 0,Y 546.139,Z 584.458,A -85,B 0,C 180,E1 -11625.505,E2 -11625.505} C_VEL
LIN {X 0,Y 548.643,Z 473.977,A -85,B 0,C 180,E1 -11627.418,E2 -11627.418} C_VEL
LIN {X 0,Y 548.687,Z 464.455,A -85,B 0,C 180,E1 -11627.598,E2 -11627.598} C_VEL
LIN {X 0,Y 546.766,Z 442.716,A -85,B 0,C 180,E1 -11628.116,E2 -11628.116} C_VEL
LIN {X 0,Y 545.597,Z 432.948,A -85,B 0,C 180,E1 -11628.398,E2 -11628.398} C_VEL
LIN {X 0,Y 543.339,Z 412.534,A -85,B 0,C 180,E1 -11629.216,E2 -11629.216} C_VEL
LIN {X 0,Y 544.538,Z 385.149,A -85,B 0,C 180,E1 -11632.351,E2 -11632.351} C_VEL
LIN {X 0,Y 545.866,Z 354.749,A -85,B 0,C 180,E1 -11635.867,E2 -11635.867} C_VEL
LIN {X 0,Y 545.92,Z 349.282,A -85,B 0,C 180,E1 -11636.51,E2 -11636.51} C_VEL
LIN {X 0,Y 542.142,Z 330.513,A -85,B 0,C 180,E1 -11638.907,E2 -11638.907} C_VEL
LIN {X 0,Y 542.107,Z 330.514,A -85,B 0,C 180,E1 -11641.989,E2 -11641.989} C_VEL
LIN {X 0,Y 542.099,Z 330.515,A -85,B 0,C 180,E1 -11644.647,E2 -11644.647} C_VEL
LIN {X 0,Y 542.083,Z 330.516,A -85,B 0,C 180,E1 -11647.395,E2 -11647.395} C_VEL
LIN {X 0,Y 542.102,Z 330.514,A -85,B 0,C 180,E1 -11650.33,E2 -11650.33} C_VEL
LIN {X 0,Y 542.132,Z 330.514,A -85,B 0,C 180,E1 -11653.653,E2 -11653.653} C_VEL
LIN {X 0,Y 542.132,Z 330.513,A -85,B 0,C 180,E1 -11656.347,E2 -11656.347} C_VEL
LIN {X 0,Y 542.117,Z 330.514,A -85,B 0,C 180,E1 -11659.757,E2 -11659.757} C_VEL
LIN {X 0,Y 542.119,Z 330.516,A -85,B 0,C 180,E1 -11662.608,E2 -11662.608} C_VEL
LIN {X 0,Y 542.131,Z 330.515,A -85,B 0,C 180,E1 -11665.355,E2 -11665.355} C_VEL
LIN {X 0,Y 542.11,Z 330.523,A -85,B 0,C 180,E1 -11668.514,E2 -11668.514} C_VEL
LIN {X 0,Y 542.127,Z 330.614,A -85,B 0,C 180,E1 -11669.098,E2 -11669.098} C_VEL
LIN {X 0,Y 546.541,Z 344.347,A -85,B 0,C 180,E1 -11671.052,E2 -11671.052} C_VEL
LIN {X 0,Y 549.529,Z 356.818,A -85,B 0,C 180,E1 -11672.686,E2 -11672.686} C_VEL
LIN {X 0,Y 549.787,Z 360.349,A -85,B 0,C 180,E1 -11673.103,E2 -11673.103} C_VEL
LIN {X 0,Y 548.39,Z 387.621,A -85,B 0,C 180,E1 -11676.075,E2 -11676.075} C_VEL
LIN {X 0,Y 547.128,Z 412.897,A -85,B 0,C 180,E1 -11678.798,E2 -11678.798} C_VEL
LIN {X 0,Y 546.095,Z 437.771,A -85,B 0,C 180,E1 -11681.488,E2 -11681.488} C_VEL
LIN {X 0,Y 546.027,Z 439.741,A -85,B 0,C 180,E1 -11681.694,E2 -11681.694} C_VEL
LIN {X 0,Y 549,Z 458.316,A -85,B 0,C 180,E1 -11682.199,E2 -11682.199} C_VEL
LIN {X 0,Y 549.471,Z 463.961,A -85,B 0,C 180,E1 -11682.329,E2 -11682.329} C_VEL
LIN {X 0,Y 547.222,Z 556.304,A -85,B 0,C 180,E1 -11683.91,E2 -11683.91} C_VEL
LIN {X 0,Y 546.644,Z 582.549,A -85,B 0,C 180,E1 -11684.374,E2 -11684.374} C_VEL
LIN {X 0,Y 546.099,Z 597.618,A -85,B 0,C 180,E1 -11684.803,E2 -11684.803} C_VEL
LIN {X 0,Y 545.544,Z 610.576,A -85,B 0,C 180,E1 -11685.311,E2 -11685.311} C_VEL
LIN {X 0,Y 544.917,Z 623.464,A -85,B 0,C 180,E1 -11685.959,E2 -11685.959} C_VEL
LIN {X 0,Y 544.134,Z 636.711,A -85,B 0,C 180,E1 -11686.792,E2 -11686.792} C_VEL
LIN {X 0,Y 543.415,Z 648.609,A -85,B 0,C 180,E1 -11687.721,E2 -11687.721} C_VEL
LIN {X 0,Y 542.766,Z 659.457,A -85,B 0,C 180,E1 -11688.751,E2 -11688.751} C_VEL
LIN {X 0,Y 542.238,Z 669.879,A -85,B 0,C 180,E1 -11689.957,E2 -11689.957} C_VEL
LIN {X 0,Y 541.644,Z 679.093,A -85,B 0,C 180,E1 -11691.26,E2 -11691.26} C_VEL
LIN {X 0,Y 541.277,Z 686.483,A -85,B 0,C 180,E1 -11692.565,E2 -11692.565} C_VEL
LIN {X 0,Y 541.051,Z 691.644,A -85,B 0,C 180,E1 -11693.682,E2 -11693.682} C_VEL
LIN {X 0,Y 540.8,Z 696.952,A -85,B 0,C 180,E1 -11695.171,E2 -11695.171} C_VEL
LIN {X 0,Y 540.731,Z 699.915,A -85,B 0,C 180,E1 -11696.287,E2 -11696.287} C_VEL
LIN {X 0,Y 540.684,Z 702.535,A -85,B 0,C 180,E1 -11697.773,E2 -11697.773} C_VEL
LIN {X 0,Y 540.613,Z 703.707,A -85,B 0,C 180,E1 -11699.258,E2 -11699.258} C_VEL
LIN {X 0,Y 540.612,Z 703.465,A -85,B 0,C 180,E1 -11700.743,E2 -11700.743} C_VEL
LIN {X 0,Y 540.682,Z 701.805,A -85,B 0,C 180,E1 -11702.228,E2 -11702.228} C_VEL
LIN {X 0,Y 540.693,Z 698.7,A -85,B 0,C 180,E1 -11703.714,E2 -11703.714} C_VEL
LIN {X 0,Y 540.827,Z 694.051,A -85,B 0,C 180,E1 -11705.202,E2 -11705.202} C_VEL
LIN {X 0,Y 540.908,Z 689.433,A -85,B 0,C 180,E1 -11706.32,E2 -11706.32} C_VEL
LIN {X 0,Y 541.161,Z 682.739,A -85,B 0,C 180,E1 -11707.624,E2 -11707.624} C_VEL
LIN {X 0,Y 541.47,Z 674.349,A -85,B 0,C 180,E1 -11708.93,E2 -11708.93} C_VEL
LIN {X 0,Y 541.857,Z 665.581,A -85,B 0,C 180,E1 -11710.05,E2 -11710.05} C_VEL
LIN {X 0,Y 542.349,Z 654.969,A -85,B 0,C 180,E1 -11711.171,E2 -11711.171} C_VEL
LIN {X 0,Y 542.826,Z 643.118,A -85,B 0,C 180,E1 -11712.199,E2 -11712.199} C_VEL
LIN {X 0,Y 543.358,Z 631.264,A -85,B 0,C 180,E1 -11713.038,E2 -11713.038} C_VEL
LIN {X 0,Y 543.959,Z 618.196,A -85,B 0,C 180,E1 -11713.782,E2 -11713.782} C_VEL
LIN {X 0,Y 544.458,Z 604.686,A -85,B 0,C 180,E1 -11714.386,E2 -11714.386} C_VEL
LIN {X 0,Y 544.847,Z 590.076,A -85,B 0,C 180,E1 -11714.875,E2 -11714.875} C_VEL
LIN {X 0,Y 545.225,Z 575.816,A -85,B 0,C 180,E1 -11715.199,E2 -11715.199} C_VEL
LIN {X 0,Y 546.847,Z 460.984,A -85,B 0,C 180,E1 -11716.99,E2 -11716.99} C_VEL
LIN {X 0,Y 544.334,Z 439.414,A -85,B 0,C 180,E1 -11717.428,E2 -11717.428} C_VEL
LIN {X 0,Y 545.452,Z 407.375,A -85,B 0,C 180,E1 -11720.876,E2 -11720.876} C_VEL
LIN {X 0,Y 546.496,Z 380.236,A -85,B 0,C 180,E1 -11723.812,E2 -11723.812} C_VEL
LIN {X 0,Y 547.418,Z 356.34,A -85,B 0,C 180,E1 -11726.404,E2 -11726.404} C_VEL
LIN {X 0,Y 547.164,Z 352.627,A -85,B 0,C 180,E1 -11726.824,E2 -11726.824} C_VEL
LIN {X 0,Y 542.173,Z 330.509,A -85,B 0,C 180,E1 -11729.478,E2 -11729.478} C_VEL
LIN {X 0,Y 542.126,Z 330.51,A -85,B 0,C 180,E1 -11731.988,E2 -11731.988} C_VEL
LIN {X 0,Y 542.164,Z 330.505,A -85,B 0,C 180,E1 -11734.643,E2 -11734.643} C_VEL
LIN {X 0,Y 542.138,Z 330.513,A -85,B 0,C 180,E1 -11737.391,E2 -11737.391} C_VEL
LIN {X 0,Y 542.126,Z 330.509,A -85,B 0,C 180,E1 -11740.333,E2 -11740.333} C_VEL
LIN {X 0,Y 542.134,Z 330.513,A -85,B 0,C 180,E1 -11743.218,E2 -11743.218} C_VEL
LIN {X 0,Y 542.157,Z 330.505,A -85,B 0,C 180,E1 -11745.761,E2 -11745.761} C_VEL
LIN {X 0,Y 542.132,Z 330.516,A -85,B 0,C 180,E1 -11748.782,E2 -11748.782} C_VEL
LIN {X 0,Y 542.105,Z 330.511,A -85,B 0,C 180,E1 -11751.669,E2 -11751.669} C_VEL
LIN {X 0,Y 542.196,Z 330.506,A -85,B 0,C 180,E1 -11754.477,E2 -11754.477} C_VEL
LIN {X 0,Y 542.125,Z 330.511,A -85,B 0,C 180,E1 -11757.135,E2 -11757.135} C_VEL
LIN {X 0,Y 542.144,Z 330.509,A -85,B 0,C 180,E1 -11759.956,E2 -11759.956} C_VEL
LIN {X 0,Y 542.159,Z 330.512,A -85,B 0,C 180,E1 -11762.283,E2 -11762.283} C_VEL
LIN {X 0,Y 542.141,Z 330.508,A -85,B 0,C 180,E1 -11765.579,E2 -11765.579} C_VEL
LIN {X 0,Y 542.176,Z 330.507,A -85,B 0,C 180,E1 -11768.463,E2 -11768.463} C_VEL
LIN {X 0,Y 542.159,Z 330.505,A -85,B 0,C 180,E1 -11771.156,E2 -11771.156} C_VEL
LIN {X 0,Y 542.157,Z 330.507,A -85,B 0,C 180,E1 -11774.013,E2 -11774.013} C_VEL
LIN {X 0,Y 541.504,Z 330.593,A -85,B 0,C 180,E1 -11774.633,E2 -11774.633} C_VEL
LIN {X 0,Y 538.652,Z 330.95,A -85,B 0,C 180,E1 -11775.64,E2 -11775.64} C_VEL
LIN {X 0,Y 536.24,Z 331.245,A -85,B 0,C 180,E1 -11776.45,E2 -11776.45} C_VEL
LIN {X 0,Y 535.216,Z 331.371,A -85,B 0,C 180,E1 -11777.076,E2 -11777.076} C_VEL
LIN {X 0,Y 535.139,Z 331.382,A -85,B 0,C 180,E1 -11777.288,E2 -11777.288} C_VEL
LIN {X 0,Y 535.172,Z 331.382,A -85,B 0,C 180,E1 -11777.593,E2 -11777.593} C_VEL
LIN {X 0,Y 540.676,Z 347.548,A -85,B 0,C 180,E1 -11777.99,E2 -11777.99} C_VEL
LIN {X 0,Y 539.834,Z 449.043,A -85,B 0,C 180,E1 -11779.345,E2 -11779.345} C_VEL
LIN {X 0,Y 539.73,Z 463.469,A -85,B 0,C 180,E1 -11779.65,E2 -11779.65} C_VEL
LIN {X 0,Y 539.446,Z 477.29,A -85,B 0,C 180,E1 -11780.093,E2 -11780.093} C_VEL
LIN {X 0,Y 539.067,Z 490.136,A -85,B 0,C 180,E1 -11780.653,E2 -11780.653} C_VEL
LIN {X 0,Y 538.659,Z 501.789,A -85,B 0,C 180,E1 -11781.3,E2 -11781.3} C_VEL
LIN {X 0,Y 538.199,Z 514.073,A -85,B 0,C 180,E1 -11782.146,E2 -11782.146} C_VEL
LIN {X 0,Y 537.578,Z 525.139,A -85,B 0,C 180,E1 -11783.078,E2 -11783.078} C_VEL
LIN {X 0,Y 536.96,Z 534.339,A -85,B 0,C 180,E1 -11784.01,E2 -11784.01} C_VEL
LIN {X 0,Y 536.424,Z 543.582,A -85,B 0,C 180,E1 -11785.131,E2 -11785.131} C_VEL
LIN {X 0,Y 535.935,Z 552.398,A -85,B 0,C 180,E1 -11786.441,E2 -11786.441} C_VEL
LIN {X 0,Y 535.332,Z 559.548,A -85,B 0,C 180,E1 -11787.751,E2 -11787.751} C_VEL
LIN {X 0,Y 534.943,Z 565.959,A -85,B 0,C 180,E1 -11789.25,E2 -11789.25} C_VEL
LIN {X 0,Y 534.628,Z 570.778,A -85,B 0,C 180,E1 -11790.751,E2 -11790.751} C_VEL
LIN {X 0,Y 534.617,Z 574.125,A -85,B 0,C 180,E1 -11792.253,E2 -11792.253} C_VEL
LIN {X 0,Y 534.572,Z 576.141,A -85,B 0,C 180,E1 -11793.757,E2 -11793.757} C_VEL
LIN {X 0,Y 534.551,Z 576.864,A -85,B 0,C 180,E1 -11795.263,E2 -11795.263} C_VEL
LIN {X 0,Y 534.643,Z 576.285,A -85,B 0,C 180,E1 -11796.772,E2 -11796.772} C_VEL
LIN {X 0,Y 534.784,Z 574.392,A -85,B 0,C 180,E1 -11798.284,E2 -11798.284} C_VEL
LIN {X 0,Y 535.09,Z 571.118,A -85,B 0,C 180,E1 -11799.798,E2 -11799.798} C_VEL
LIN {X 0,Y 535.497,Z 566.369,A -85,B 0,C 180,E1 -11801.315,E2 -11801.315} C_VEL
LIN {X 0,Y 536.035,Z 559.99,A -85,B 0,C 180,E1 -11802.835,E2 -11802.835} C_VEL
LIN {X 0,Y 536.641,Z 552.858,A -85,B 0,C 180,E1 -11804.166,E2 -11804.166} C_VEL
LIN {X 0,Y 537.368,Z 544.267,A -85,B 0,C 180,E1 -11805.46,E2 -11805.46} C_VEL
LIN {X 0,Y 538.09,Z 534.62,A -85,B 0,C 180,E1 -11806.641,E2 -11806.641} C_VEL
LIN {X 0,Y 538.755,Z 524.214,A -85,B 0,C 180,E1 -11807.692,E2 -11807.692} C_VEL
LIN {X 0,Y 539.449,Z 512.941,A -85,B 0,C 180,E1 -11808.627,E2 -11808.627} C_VEL
LIN {X 0,Y 540.115,Z 501.378,A -85,B 0,C 180,E1 -11809.41,E2 -11809.41} C_VEL
LIN {X 0,Y 540.657,Z 489.104,A -85,B 0,C 180,E1 -11810.079,E2 -11810.079} C_VEL
LIN {X 0,Y 540.936,Z 478.208,A -85,B 0,C 180,E1 -11810.558,E2 -11810.558} C_VEL
LIN {X 0,Y 541.225,Z 464.24,A -85,B 0,C 180,E1 -11811.015,E2 -11811.015} C_VEL
LIN {X 0,Y 541.349,Z 450.654,A -85,B 0,C 180,E1 -11811.314,E2 -11811.314} C_VEL
LIN {X 0,Y 542.398,Z 350.616,A -85,B 0,C 180,E1 -11812.662,E2 -11812.662} C_VEL
LIN {X 0,Y 540.853,Z 346.097,A -85,B 0,C 180,E1 -11812.785,E2 -11812.785} C_VEL
LIN {X 0,Y 535.122,Z 331.622,A -85,B 0,C 180,E1 -11813.215,E2 -11813.215} C_VEL
LIN {X 0,Y 535.086,Z 331.398,A -85,B 0,C 180,E1 -11813.272,E2 -11813.272} C_VEL
LIN {X 0,Y 535.078,Z 331.395,A -85,B 0,C 180,E1 -11816.429,E2 -11816.429} C_VEL
LIN {X 0,Y 535.094,Z 331.39,A -85,B 0,C 180,E1 -11818.969,E2 -11818.969} C_VEL
LIN {X 0,Y 535.066,Z 331.39,A -85,B 0,C 180,E1 -11821.689,E2 -11821.689} C_VEL
LIN {X 0,Y 535.047,Z 331.397,A -85,B 0,C 180,E1 -11824.436,E2 -11824.436} C_VEL
LIN {X 0,Y 535.052,Z 331.391,A -85,B 0,C 180,E1 -11827.027,E2 -11827.027} C_VEL
LIN {X 0,Y 535.072,Z 331.393,A -85,B 0,C 180,E1 -11829.9,E2 -11829.9} C_VEL
LIN {X 0,Y 535.042,Z 331.394,A -85,B 0,C 180,E1 -11832.903,E2 -11832.903} C_VEL
LIN {X 0,Y 535.102,Z 331.382,A -85,B 0,C 180,E1 -11835.02,E2 -11835.02} C_VEL
LIN {X 0,Y 535.081,Z 331.391,A -85,B 0,C 180,E1 -11838.259,E2 -11838.259} C_VEL
LIN {X 0,Y 535.032,Z 331.389,A -85,B 0,C 180,E1 -11841.068,E2 -11841.068} C_VEL
LIN {X 0,Y 535.069,Z 331.376,A -85,B 0,C 180,E1 -11844.256,E2 -11844.256} C_VEL
LIN {X 0,Y 535.068,Z 331.386,A -85,B 0,C 180,E1 -11846.91,E2 -11846.91} C_VEL
LIN {X 0,Y 535.081,Z 331.386,A -85,B 0,C 180,E1 -11849.766,E2 -11849.766} C_VEL
LIN {X 0,Y 535.089,Z 331.383,A -85,B 0,C 180,E1 -11852.731,E2 -11852.731} C_VEL
LIN {X 0,Y 535.074,Z 331.385,A -85,B 0,C 180,E1 -11855.235,E2 -11855.235} C_VEL
LIN {X 0,Y 535.119,Z 331.377,A -85,B 0,C 180,E1 -11858.499,E2 -11858.499} C_VEL
LIN {X 0,Y 535.112,Z 331.388,A -85,B 0,C 180,E1 -11860.898,E2 -11860.898} C_VEL
LIN {X 0,Y 535.102,Z 331.409,A -85,B 0,C 180,E1 -11861.941,E2 -11861.941} C_VEL
LIN {X 0,Y 539.73,Z 346.684,A -85,B 0,C 180,E1 -11862.309,E2 -11862.309} C_VEL
LIN {X 0,Y 538.319,Z 451.217,A -85,B 0,C 180,E1 -11863.973,E2 -11863.973} C_VEL
LIN {X 0,Y 538.162,Z 466.124,A -85,B 0,C 180,E1 -11864.367,E2 -11864.367} C_VEL
LIN {X 0,Y 537.888,Z 480.485,A -85,B 0,C 180,E1 -11864.903,E2 -11864.903} C_VEL
LIN {X 0,Y 537.514,Z 493.996,A -85,B 0,C 180,E1 -11865.568,E2 -11865.568} C_VEL
LIN {X 0,Y 537.106,Z 506.246,A -85,B 0,C 180,E1 -11866.327,E2 -11866.327} C_VEL
LIN {X 0,Y 536.637,Z 518.689,A -85,B 0,C 180,E1 -11867.275,E2 -11867.275} C_VEL
LIN {X 0,Y 536.186,Z 529.251,A -85,B 0,C 180,E1 -11868.251,E2 -11868.251} C_VEL
LIN {X 0,Y 535.904,Z 538.424,A -85,B 0,C 180,E1 -11869.266,E2 -11869.266} C_VEL
LIN {X 0,Y 535.446,Z 547.039,A -85,B 0,C 180,E1 -11870.399,E2 -11870.399} C_VEL
LIN {X 0,Y 535.113,Z 555.25,A -85,B 0,C 180,E1 -11871.721,E2 -11871.721} C_VEL
LIN {X 0,Y 534.874,Z 561.01,A -85,B 0,C 180,E1 -11872.853,E2 -11872.853} C_VEL
LIN {X 0,Y 534.643,Z 567.026,A -85,B 0,C 180,E1 -11874.361,E2 -11874.361} C_VEL
LIN {X 0,Y 534.501,Z 570.494,A -85,B 0,C 180,E1 -11875.49,E2 -11875.49} C_VEL
LIN {X 0,Y 534.576,Z 573.728,A -85,B 0,C 180,E1 -11876.995,E2 -11876.995} C_VEL
LIN {X 0,Y 534.471,Z 575.565,A -85,B 0,C 180,E1 -11878.498,E2 -11878.498} C_VEL
LIN {X 0,Y 534.399,Z 576.02,A -85,B 0,C 180,E1 -11880,E2 -11880} C_VEL
LIN {X 0,Y 534.532,Z 575.046,A -85,B 0,C 180,E1 -11881.502,E2 -11881.502} C_VEL
LIN {X 0,Y 534.941,Z 572.596,A -85,B 0,C 180,E1 -11883.002,E2 -11883.002} C_VEL
LIN {X 0,Y 535.428,Z 568.676,A -85,B 0,C 180,E1 -11884.502,E2 -11884.502} C_VEL
LIN {X 0,Y 535.585,Z 563.242,A -85,B 0,C 180,E1 -11886.005,E2 -11886.005} C_VEL
LIN {X 0,Y 536.282,Z 556.907,A -85,B 0,C 180,E1 -11887.316,E2 -11887.316} C_VEL
LIN {X 0,Y 536.858,Z 548.991,A -85,B 0,C 180,E1 -11888.629,E2 -11888.629} C_VEL
LIN {X 0,Y 537.397,Z 540.693,A -85,B 0,C 180,E1 -11889.755,E2 -11889.755} C_VEL
LIN {X 0,Y 538.02,Z 530.659,A -85,B 0,C 180,E1 -11890.881,E2 -11890.881} C_VEL
LIN {X 0,Y 538.627,Z 520.549,A -85,B 0,C 180,E1 -11891.819,E2 -11891.819} C_VEL
LIN {X 0,Y 539.284,Z 509.573,A -85,B 0,C 180,E1 -11892.661,E2 -11892.661} C_VEL
LIN {X 0,Y 539.929,Z 497.194,A -85,B 0,C 180,E1 -11893.432,E2 -11893.432} C_VEL
LIN {X 0,Y 540.304,Z 483.446,A -85,B 0,C 180,E1 -11894.116,E2 -11894.116} C_VEL
LIN {X 0,Y 540.644,Z 469.719,A -85,B 0,C 180,E1 -11894.633,E2 -11894.633} C_VEL
LIN {X 0,Y 540.861,Z 455.534,A -85,B 0,C 180,E1 -11895.011,E2 -11895.011} C_VEL
LIN {X 0,Y 542.574,Z 374.188,A -85,B 0,C 180,E1 -11896.429,E2 -11896.429} C_VEL
LIN {X 0,Y 543.097,Z 349.872,A -85,B 0,C 180,E1 -11896.874,E2 -11896.874} C_VEL
LIN {X 0,Y 537.357,Z 336.759,A -85,B 0,C 180,E1 -11897.438,E2 -11897.438} C_VEL
LIN {X 0,Y 535.297,Z 332.152,A -85,B 0,C 180,E1 -11897.645,E2 -11897.645} C_VEL
LIN {X 0,Y 535.149,Z 331.387,A -85,B 0,C 180,E1 -11897.697,E2 -11897.697} C_VEL
LIN {X 0,Y 535.137,Z 331.387,A -85,B 0,C 180,E1 -11900.696,E2 -11900.696} C_VEL
LIN {X 0,Y 535.1,Z 331.393,A -85,B 0,C 180,E1 -11903.94,E2 -11903.94} C_VEL
LIN {X 0,Y 535.087,Z 331.393,A -85,B 0,C 180,E1 -11906.428,E2 -11906.428} C_VEL
LIN {X 0,Y 535.101,Z 331.387,A -85,B 0,C 180,E1 -11908.968,E2 -11908.968} C_VEL
LIN {X 0,Y 535.078,Z 331.392,A -85,B 0,C 180,E1 -11911.692,E2 -11911.692} C_VEL
LIN {X 0,Y 535.106,Z 331.383,A -85,B 0,C 180,E1 -11914.446,E2 -11914.446} C_VEL
LIN {X 0,Y 535.103,Z 331.383,A -85,B 0,C 180,E1 -11917.023,E2 -11917.023} C_VEL
LIN {X 0,Y 535.074,Z 331.385,A -85,B 0,C 180,E1 -11919.899,E2 -11919.899} C_VEL
LIN {X 0,Y 535.088,Z 331.386,A -85,B 0,C 180,E1 -11922.898,E2 -11922.898} C_VEL
LIN {X 0,Y 535.098,Z 331.383,A -85,B 0,C 180,E1 -11926.07,E2 -11926.07} C_VEL
LIN {X 0,Y 535.059,Z 331.395,A -85,B 0,C 180,E1 -11929.114,E2 -11929.114} C_VEL
LIN {X 0,Y 535.04,Z 331.394,A -85,B 0,C 180,E1 -11932.026,E2 -11932.026} C_VEL
LIN {X 0,Y 535.045,Z 331.391,A -85,B 0,C 180,E1 -11934.829,E2 -11934.829} C_VEL
LIN {X 0,Y 535.048,Z 331.395,A -85,B 0,C 180,E1 -11937.538,E2 -11937.538} C_VEL
LIN {X 0,Y 535.118,Z 331.501,A -85,B 0,C 180,E1 -11940.082,E2 -11940.082} C_VEL
LIN {X 0,Y 538.838,Z 347.847,A -85,B 0,C 180,E1 -11942.326,E2 -11942.326} C_VEL
LIN {X 0,Y 540.108,Z 355.616,A -85,B 0,C 180,E1 -11943.346,E2 -11943.346} C_VEL
LIN {X 0,Y 538.919,Z 375.238,A -85,B 0,C 180,E1 -11945.701,E2 -11945.701} C_VEL
LIN {X 0,Y 537.514,Z 401.337,A -85,B 0,C 180,E1 -11948.8,E2 -11948.8} C_VEL
LIN {X 0,Y 536.39,Z 426.505,A -85,B 0,C 180,E1 -11951.735,E2 -11951.735} C_VEL
LIN {X 0,Y 540.449,Z 458.786,A -85,B 0,C 180,E1 -11952.33,E2 -11952.33} C_VEL
LIN {X 0,Y 541.194,Z 468.681,A -85,B 0,C 180,E1 -11952.492,E2 -11952.492} C_VEL
LIN {X 0,Y 540.092,Z 566.312,A -85,B 0,C 180,E1 -11953.813,E2 -11953.813} C_VEL
LIN {X 0,Y 539.487,Z 580.675,A -85,B 0,C 180,E1 -11954.153,E2 -11954.153} C_VEL
LIN {X 0,Y 538.702,Z 594.607,A -85,B 0,C 180,E1 -11954.637,E2 -11954.637} C_VEL
LIN {X 0,Y 537.817,Z 608.492,A -85,B 0,C 180,E1 -11955.288,E2 -11955.288} C_VEL
LIN {X 0,Y 537.01,Z 620.962,A -85,B 0,C 180,E1 -11956.036,E2 -11956.036} C_VEL
LIN {X 0,Y 536.062,Z 633.566,A -85,B 0,C 180,E1 -11956.974,E2 -11956.974} C_VEL
LIN {X 0,Y 535.423,Z 649.762,A -85,B 0,C 180,E1 -11958.205,E2 -11958.205} C_VEL
LIN {X 0,Y 534.915,Z 661.248,A -85,B 0,C 180,E1 -11959.274,E2 -11959.274} C_VEL
LIN {X 0,Y 534.525,Z 671.052,A -85,B 0,C 180,E1 -11960.382,E2 -11960.382} C_VEL
LIN {X 0,Y 534.168,Z 679.376,A -85,B 0,C 180,E1 -11961.517,E2 -11961.517} C_VEL
LIN {X 0,Y 533.944,Z 687.316,A -85,B 0,C 180,E1 -11962.841,E2 -11962.841} C_VEL
LIN {X 0,Y 533.82,Z 692.803,A -85,B 0,C 180,E1 -11963.974,E2 -11963.974} C_VEL
LIN {X 0,Y 533.734,Z 697.25,A -85,B 0,C 180,E1 -11965.106,E2 -11965.106} C_VEL
LIN {X 0,Y 533.665,Z 700.76,A -85,B 0,C 180,E1 -11966.237,E2 -11966.237} C_VEL
LIN {X 0,Y 533.666,Z 704.002,A -85,B 0,C 180,E1 -11967.743,E2 -11967.743} C_VEL
LIN {X 0,Y 533.607,Z 705.767,A -85,B 0,C 180,E1 -11969.248,E2 -11969.248} C_VEL
LIN {X 0,Y 533.606,Z 706.087,A -85,B 0,C 180,E1 -11970.752,E2 -11970.752} C_VEL
LIN {X 0,Y 533.669,Z 704.97,A -85,B 0,C 180,E1 -11972.257,E2 -11972.257} C_VEL
LIN {X 0,Y 533.676,Z 702.404,A -85,B 0,C 180,E1 -11973.763,E2 -11973.763} C_VEL
LIN {X 0,Y 533.815,Z 698.277,A -85,B 0,C 180,E1 -11975.27,E2 -11975.27} C_VEL
LIN {X 0,Y 534.013,Z 692.495,A -85,B 0,C 180,E1 -11976.779,E2 -11976.779} C_VEL
LIN {X 0,Y 534.338,Z 685.952,A -85,B 0,C 180,E1 -11978.101,E2 -11978.101} C_VEL
LIN {X 0,Y 534.749,Z 677.785,A -85,B 0,C 180,E1 -11979.423,E2 -11979.423} C_VEL
LIN {X 0,Y 535.292,Z 669.212,A -85,B 0,C 180,E1 -11980.556,E2 -11980.556} C_VEL
LIN {X 0,Y 535.721,Z 660.71,A -85,B 0,C 180,E1 -11981.501,E2 -11981.501} C_VEL
LIN {X 0,Y 536.428,Z 649.589,A -85,B 0,C 180,E1 -11982.538,E2 -11982.538} C_VEL
LIN {X 0,Y 537.118,Z 637.161,A -85,B 0,C 180,E1 -11983.48,E2 -11983.48} C_VEL
LIN {X 0,Y 537.838,Z 624.908,A -85,B 0,C 180,E1 -11984.23,E2 -11984.23} C_VEL
LIN {X 0,Y 538.425,Z 611.499,A -85,B 0,C 180,E1 -11984.888,E2 -11984.888} C_VEL
LIN {X 0,Y 539.074,Z 597.017,A -85,B 0,C 180,E1 -11985.424,E2 -11985.424} C_VEL
LIN {X 0,Y 539.507,Z 582.577,A -85,B 0,C 180,E1 -11985.797,E2 -11985.797} C_VEL
LIN {X 0,Y 542.058,Z 478.095,A -85,B 0,C 180,E1 -11987.643,E2 -11987.643} C_VEL
LIN {X 0,Y 542.234,Z 465.478,A -85,B 0,C 180,E1 -11987.885,E2 -11987.885} C_VEL
LIN {X 0,Y 540.319,Z 443.306,A -85,B 0,C 180,E1 -11988.429,E2 -11988.429} C_VEL
LIN {X 0,Y 539.103,Z 433.21,A -85,B 0,C 180,E1 -11988.732,E2 -11988.732} C_VEL
LIN {X 0,Y 536.477,Z 409.215,A -85,B 0,C 180,E1 -11989.745,E2 -11989.745} C_VEL
LIN {X 0,Y 537.651,Z 382.871,A -85,B 0,C 180,E1 -11992.804,E2 -11992.804} C_VEL
LIN {X 0,Y 538.956,Z 355.45,A -85,B 0,C 180,E1 -11996.016,E2 -11996.016} C_VEL
LIN {X 0,Y 538.929,Z 350.255,A -85,B 0,C 180,E1 -11996.64,E2 -11996.64} C_VEL
LIN {X 0,Y 535.099,Z 331.391,A -85,B 0,C 180,E1 -11999.089,E2 -11999.089} C_VEL
LIN {X 0,Y 535.061,Z 331.395,A -85,B 0,C 180,E1 -12001.689,E2 -12001.689} C_VEL
LIN {X 0,Y 535.041,Z 331.394,A -85,B 0,C 180,E1 -12004.436,E2 -12004.436} C_VEL
LIN {X 0,Y 535.046,Z 331.396,A -85,B 0,C 180,E1 -12007.028,E2 -12007.028} C_VEL
LIN {X 0,Y 535.067,Z 331.391,A -85,B 0,C 180,E1 -12009.9,E2 -12009.9} C_VEL
LIN {X 0,Y 535.044,Z 331.397,A -85,B 0,C 180,E1 -12012.902,E2 -12012.902} C_VEL
LIN {X 0,Y 535.098,Z 331.392,A -85,B 0,C 180,E1 -12015.02,E2 -12015.02} C_VEL
LIN {X 0,Y 535.049,Z 331.395,A -85,B 0,C 180,E1 -12018.114,E2 -12018.114} C_VEL
LIN {X 0,Y 535.032,Z 331.4,A -85,B 0,C 180,E1 -12021.068,E2 -12021.068} C_VEL
LIN {X 0,Y 535.093,Z 331.39,A -85,B 0,C 180,E1 -12023.91,E2 -12023.91} C_VEL
LIN {X 0,Y 535.065,Z 331.397,A -85,B 0,C 180,E1 -12026.91,E2 -12026.91} C_VEL
LIN {X 0,Y 535.101,Z 331.589,A -85,B 0,C 180,E1 -12028.591,E2 -12028.591} C_VEL
LIN {X 0,Y 540.003,Z 346.47,A -85,B 0,C 180,E1 -12030.79,E2 -12030.79} C_VEL
LIN {X 0,Y 542.793,Z 357.838,A -85,B 0,C 180,E1 -12032.318,E2 -12032.318} C_VEL
LIN {X 0,Y 543.347,Z 361.735,A -85,B 0,C 180,E1 -12032.811,E2 -12032.811} C_VEL
LIN {X 0,Y 541.882,Z 388.605,A -85,B 0,C 180,E1 -12035.77,E2 -12035.77} C_VEL
LIN {X 0,Y 540.524,Z 413.809,A -85,B 0,C 180,E1 -12038.526,E2 -12038.526} C_VEL
LIN {X 0,Y 539.382,Z 439.895,A -85,B 0,C 180,E1 -12041.359,E2 -12041.359} C_VEL
LIN {X 0,Y 542.236,Z 457.197,A -85,B 0,C 180,E1 -12041.853,E2 -12041.853} C_VEL
LIN {X 0,Y 542.957,Z 464.701,A -85,B 0,C 180,E1 -12042.037,E2 -12042.037} C_VEL
LIN {X 0,Y 540.552,Z 557.872,A -85,B 0,C 180,E1 -12043.675,E2 -12043.675} C_VEL
LIN {X 0,Y 539.967,Z 582.72,A -85,B 0,C 180,E1 -12044.126,E2 -12044.126} C_VEL
LIN {X 0,Y 539.38,Z 597.694,A -85,B 0,C 180,E1 -12044.561,E2 -12044.561} C_VEL
LIN {X 0,Y 538.717,Z 611.613,A -85,B 0,C 180,E1 -12045.12,E2 -12045.12} C_VEL
LIN {X 0,Y 537.998,Z 625.905,A -85,B 0,C 180,E1 -12045.871,E2 -12045.871} C_VEL
LIN {X 0,Y 537.202,Z 638.603,A -85,B 0,C 180,E1 -12046.714,E2 -12046.714} C_VEL
LIN {X 0,Y 536.464,Z 650.156,A -85,B 0,C 180,E1 -12047.655,E2 -12047.655} C_VEL
LIN {X 0,Y 535.777,Z 660.684,A -85,B 0,C 180,E1 -12048.691,E2 -12048.691} C_VEL
LIN {X 0,Y 535.243,Z 670.231,A -85,B 0,C 180,E1 -12049.824,E2 -12049.824} C_VEL
LIN {X 0,Y 534.608,Z 679.378,A -85,B 0,C 180,E1 -12051.144,E2 -12051.144} C_VEL
LIN {X 0,Y 534.221,Z 686.711,A -85,B 0,C 180,E1 -12052.466,E2 -12052.466} C_VEL
LIN {X 0,Y 533.98,Z 691.836,A -85,B 0,C 180,E1 -12053.598,E2 -12053.598} C_VEL
LIN {X 0,Y 533.73,Z 697.099,A -85,B 0,C 180,E1 -12055.107,E2 -12055.107} C_VEL
LIN {X 0,Y 533.666,Z 700.043,A -85,B 0,C 180,E1 -12056.237,E2 -12056.237} C_VEL
LIN {X 0,Y 533.596,Z 702.606,A -85,B 0,C 180,E1 -12057.743,E2 -12057.743} C_VEL
LIN {X 0,Y 533.536,Z 703.735,A -85,B 0,C 180,E1 -12059.248,E2 -12059.248} C_VEL
LIN {X 0,Y 533.535,Z 703.447,A -85,B 0,C 180,E1 -12060.752,E2 -12060.752} C_VEL
LIN {X 0,Y 533.594,Z 701.737,A -85,B 0,C 180,E1 -12062.257,E2 -12062.257} C_VEL
LIN {X 0,Y 533.618,Z 698.575,A -85,B 0,C 180,E1 -12063.763,E2 -12063.763} C_VEL
LIN {X 0,Y 533.68,Z 695.154,A -85,B 0,C 180,E1 -12064.894,E2 -12064.894} C_VEL
LIN {X 0,Y 533.792,Z 690.82,A -85,B 0,C 180,E1 -12066.026,E2 -12066.026} C_VEL
LIN {X 0,Y 534.019,Z 684.452,A -85,B 0,C 180,E1 -12067.348,E2 -12067.348} C_VEL
LIN {X 0,Y 534.284,Z 676.492,A -85,B 0,C 180,E1 -12068.671,E2 -12068.671} C_VEL
LIN {X 0,Y 534.67,Z 668.158,A -85,B 0,C 180,E1 -12069.806,E2 -12069.806} C_VEL
LIN {X 0,Y 535.191,Z 657.404,A -85,B 0,C 180,E1 -12071.013,E2 -12071.013} C_VEL
LIN {X 0,Y 535.667,Z 645.745,A -85,B 0,C 180,E1 -12072.077,E2 -12072.077} C_VEL
LIN {X 0,Y 536.264,Z 633.038,A -85,B 0,C 180,E1 -12073.021,E2 -12073.021} C_VEL
LIN {X 0,Y 536.86,Z 620.487,A -85,B 0,C 180,E1 -12073.775,E2 -12073.775} C_VEL
LIN {X 0,Y 537.419,Z 606.516,A -85,B 0,C 180,E1 -12074.434,E2 -12074.434} C_VEL
LIN {X 0,Y 537.85,Z 591.75,A -85,B 0,C 180,E1 -12074.953,E2 -12074.953} C_VEL
LIN {X 0,Y 538.187,Z 577.289,A -85,B 0,C 180,E1 -12075.303,E2 -12075.303} C_VEL
LIN {X 0,Y 539.922,Z 461.387,A -85,B 0,C 180,E1 -12077.154,E2 -12077.154} C_VEL
LIN {X 0,Y 537.367,Z 439.571,A -85,B 0,C 180,E1 -12077.59,E2 -12077.59} C_VEL
LIN {X 0,Y 538.484,Z 408.549,A -85,B 0,C 180,E1 -12080.96,E2 -12080.96} C_VEL
LIN {X 0,Y 539.565,Z 381.261,A -85,B 0,C 180,E1 -12083.934,E2 -12083.934} C_VEL
LIN {X 0,Y 540.553,Z 356.855,A -85,B 0,C 180,E1 -12086.607,E2 -12086.607} C_VEL
LIN {X 0,Y 539.672,Z 351.613,A -85,B 0,C 180,E1 -12087.222,E2 -12087.222} C_VEL
LIN {X 0,Y 535.439,Z 332.851,A -85,B 0,C 180,E1 -12089.485,E2 -12089.485} C_VEL
LIN {X 0,Y 535.109,Z 331.389,A -85,B 0,C 180,E1 -12089.667,E2 -12089.667} C_VEL
LIN {X 0,Y 535.077,Z 331.388,A -85,B 0,C 180,E1 -12092.46,E2 -12092.46} C_VEL
LIN {X 0,Y 535.123,Z 331.388,A -85,B 0,C 180,E1 -12095.165,E2 -12095.165} C_VEL
LIN {X 0,Y 535.086,Z 331.386,A -85,B 0,C 180,E1 -12097.97,E2 -12097.97} C_VEL
LIN {X 0,Y 535.097,Z 331.39,A -85,B 0,C 180,E1 -12100.882,E2 -12100.882} C_VEL
LIN {X 0,Y 535.129,Z 331.38,A -85,B 0,C 180,E1 -12103.953,E2 -12103.953} C_VEL
LIN {X 0,Y 535.102,Z 331.384,A -85,B 0,C 180,E1 -12106.071,E2 -12106.071} C_VEL
LIN {X 0,Y 535.103,Z 331.388,A -85,B 0,C 180,E1 -12109.119,E2 -12109.119} C_VEL
LIN {X 0,Y 535.086,Z 331.386,A -85,B 0,C 180,E1 -12112.03,E2 -12112.03} C_VEL
LIN {X 0,Y 535.122,Z 331.386,A -85,B 0,C 180,E1 -12114.835,E2 -12114.835} C_VEL
LIN {X 0,Y 535.068,Z 331.388,A -85,B 0,C 180,E1 -12117.539,E2 -12117.539} C_VEL
LIN {X 0,Y 535.097,Z 331.389,A -85,B 0,C 180,E1 -12120.17,E2 -12120.17} C_VEL
LIN {X 0,Y 535.106,Z 331.385,A -85,B 0,C 180,E1 -12122.888,E2 -12122.888} C_VEL
LIN {X 0,Y 535.098,Z 331.39,A -85,B 0,C 180,E1 -12126.059,E2 -12126.059} C_VEL
LIN {X 0,Y 535.137,Z 331.38,A -85,B 0,C 180,E1 -12129.304,E2 -12129.304} C_VEL
LIN {X 0,Y 535.102,Z 331.387,A -85,B 0,C 180,E1 -12131.69,E2 -12131.69} C_VEL
LIN {X 0,Y 535.129,Z 331.388,A -85,B 0,C 180,E1 -12134.046,E2 -12134.046} C_VEL
LIN {X 0,Y 535.167,Z 331.379,A -85,B 0,C 180,E1 -12136.374,E2 -12136.374} C_VEL
LIN {X 0,Y 535.139,Z 331.382,A -85,B 0,C 180,E1 -12137.288,E2 -12137.288} C_VEL
LIN {X 0,Y 535.875,Z 331.643,A -85,B 0,C 180,E1 -12137.496,E2 -12137.496} C_VEL
LIN {X 0,Y 537.98,Z 332.43,A -85,B 0,C 180,E1 -12137.684,E2 -12137.684} C_VEL
LIN {X 0,Y 542.903,Z 334.706,A -85,B 0,C 180,E1 -12137.884,E2 -12137.884} C_VEL
LIN {X 0,Y 546.783,Z 337.675,A -85,B 0,C 180,E1 -12138.041,E2 -12138.041} C_VEL
LIN {X 0,Y 548.843,Z 340.758,A -85,B 0,C 180,E1 -12138.145,E2 -12138.145} C_VEL
LIN {X 0,Y 549.256,Z 343.457,A -85,B 0,C 180,E1 -12138.191,E2 -12138.191} C_VEL
LIN {X 0,Y 548.173,Z 346.699,A -85,B 0,C 180,E1 -12138.187,E2 -12138.187} C_VEL
LIN {X 0,Y 545.727,Z 349.769,A -85,B 0,C 180,E1 -12138.157,E2 -12138.157} C_VEL
LIN {X 0,Y 536.721,Z 357.868,A -85,B 0,C 180,E1 -12138.009,E2 -12138.009} C_VEL
LIN {X 0,Y 534.846,Z 361.266,A -85,B 0,C 180,E1 -12137.998,E2 -12137.998} C_VEL
LIN {X 0,Y 534.374,Z 362.821,A -85,B 0,C 180,E1 -12138.003,E2 -12138.003} C_VEL
LIN {X 0,Y 533.683,Z 362.577,A -85,B 0,C 180,E1 -12137.98,E2 -12137.98} C_VEL
LIN {X 0,Y 532.995,Z 449.592,A -85,B 0,C 180,E1 -12139.159,E2 -12139.159} C_VEL
LIN {X 0,Y 532.874,Z 463.209,A -85,B 0,C 180,E1 -12139.444,E2 -12139.444} C_VEL
LIN {X 0,Y 532.628,Z 476.679,A -85,B 0,C 180,E1 -12139.87,E2 -12139.87} C_VEL
LIN {X 0,Y 532.231,Z 489.851,A -85,B 0,C 180,E1 -12140.436,E2 -12140.436} C_VEL
LIN {X 0,Y 531.746,Z 503.157,A -85,B 0,C 180,E1 -12141.179,E2 -12141.179} C_VEL
LIN {X 0,Y 531.269,Z 515.412,A -85,B 0,C 180,E1 -12142.043,E2 -12142.043} C_VEL
LIN {X 0,Y 530.607,Z 526.365,A -85,B 0,C 180,E1 -12142.986,E2 -12142.986} C_VEL
LIN {X 0,Y 529.863,Z 537.134,A -85,B 0,C 180,E1 -12144.12,E2 -12144.12} C_VEL
LIN {X 0,Y 529.274,Z 546.026,A -85,B 0,C 180,E1 -12145.256,E2 -12145.256} C_VEL
LIN {X 0,Y 528.806,Z 554.515,A -85,B 0,C 180,E1 -12146.583,E2 -12146.583} C_VEL
LIN {X 0,Y 528.3,Z 560.52,A -85,B 0,C 180,E1 -12147.721,E2 -12147.721} C_VEL
LIN {X 0,Y 527.898,Z 566.888,A -85,B 0,C 180,E1 -12149.24,E2 -12149.24} C_VEL
LIN {X 0,Y 527.587,Z 571.665,A -85,B 0,C 180,E1 -12150.761,E2 -12150.761} C_VEL
LIN {X 0,Y 527.562,Z 574.975,A -85,B 0,C 180,E1 -12152.283,E2 -12152.283} C_VEL
LIN {X 0,Y 527.504,Z 576.956,A -85,B 0,C 180,E1 -12153.807,E2 -12153.807} C_VEL
LIN {X 0,Y 527.522,Z 577.633,A -85,B 0,C 180,E1 -12155.333,E2 -12155.333} C_VEL
LIN {X 0,Y 527.594,Z 577.014,A -85,B 0,C 180,E1 -12156.863,E2 -12156.863} C_VEL
LIN {X 0,Y 527.75,Z 575.079,A -85,B 0,C 180,E1 -12158.395,E2 -12158.395} C_VEL
LIN {X 0,Y 528.111,Z 571.764,A -85,B 0,C 180,E1 -12159.929,E2 -12159.929} C_VEL
LIN {X 0,Y 528.527,Z 566.975,A -85,B 0,C 180,E1 -12161.466,E2 -12161.466} C_VEL
LIN {X 0,Y 529.111,Z 560.552,A -85,B 0,C 180,E1 -12163.006,E2 -12163.006} C_VEL
LIN {X 0,Y 529.72,Z 553.373,A -85,B 0,C 180,E1 -12164.355,E2 -12164.355} C_VEL
LIN {X 0,Y 530.501,Z 544.703,A -85,B 0,C 180,E1 -12165.665,E2 -12165.665} C_VEL
LIN {X 0,Y 531.254,Z 534.981,A -85,B 0,C 180,E1 -12166.862,E2 -12166.862} C_VEL
LIN {X 0,Y 531.984,Z 524.491,A -85,B 0,C 180,E1 -12167.925,E2 -12167.925} C_VEL
LIN {X 0,Y 532.692,Z 513.118,A -85,B 0,C 180,E1 -12168.872,E2 -12168.872} C_VEL
LIN {X 0,Y 533.386,Z 501.415,A -85,B 0,C 180,E1 -12169.665,E2 -12169.665} C_VEL
LIN {X 0,Y 533.943,Z 488.952,A -85,B 0,C 180,E1 -12170.343,E2 -12170.343} C_VEL
LIN {X 0,Y 534.251,Z 476.854,A -85,B 0,C 180,E1 -12170.862,E2 -12170.862} C_VEL
LIN {X 0,Y 534.504,Z 462.718,A -85,B 0,C 180,E1 -12171.308,E2 -12171.308} C_VEL
LIN {X 0,Y 534.668,Z 448.615,A -85,B 0,C 180,E1 -12171.593,E2 -12171.593} C_VEL
LIN {X 0,Y 535.699,Z 351.556,A -85,B 0,C 180,E1 -12172.912,E2 -12172.912} C_VEL
LIN {X 0,Y 528.109,Z 332.683,A -85,B 0,C 180,E1 -12173.489,E2 -12173.489} C_VEL
LIN {X 0,Y 528.049,Z 332.274,A -85,B 0,C 180,E1 -12173.535,E2 -12173.535} C_VEL
LIN {X 0,Y 528.031,Z 332.274,A -85,B 0,C 180,E1 -12176.809,E2 -12176.809} C_VEL
LIN {X 0,Y 528.056,Z 332.265,A -85,B 0,C 180,E1 -12179.393,E2 -12179.393} C_VEL
LIN {X 0,Y 528.003,Z 332.274,A -85,B 0,C 180,E1 -12182.049,E2 -12182.049} C_VEL
LIN {X 0,Y 527.999,Z 332.272,A -85,B 0,C 180,E1 -12184.781,E2 -12184.781} C_VEL
LIN {X 0,Y 528.001,Z 332.271,A -85,B 0,C 180,E1 -12187.607,E2 -12187.607} C_VEL
LIN {X 0,Y 528.014,Z 332.273,A -85,B 0,C 180,E1 -12190.543,E2 -12190.543} C_VEL
LIN {X 0,Y 528.044,Z 332.268,A -85,B 0,C 180,E1 -12193.613,E2 -12193.613} C_VEL
LIN {X 0,Y 528.056,Z 332.267,A -85,B 0,C 180,E1 -12196.389,E2 -12196.389} C_VEL
LIN {X 0,Y 528.016,Z 332.266,A -85,B 0,C 180,E1 -12199.125,E2 -12199.125} C_VEL
LIN {X 0,Y 527.992,Z 332.269,A -85,B 0,C 180,E1 -12201.509,E2 -12201.509} C_VEL
LIN {X 0,Y 528.022,Z 332.253,A -85,B 0,C 180,E1 -12204.29,E2 -12204.29} C_VEL
LIN {X 0,Y 528.014,Z 332.265,A -85,B 0,C 180,E1 -12207.051,E2 -12207.051} C_VEL
LIN {X 0,Y 528.036,Z 332.263,A -85,B 0,C 180,E1 -12209.73,E2 -12209.73} C_VEL
LIN {X 0,Y 528.043,Z 332.261,A -85,B 0,C 180,E1 -12212.717,E2 -12212.717} C_VEL
LIN {X 0,Y 528.024,Z 332.27,A -85,B 0,C 180,E1 -12215.718,E2 -12215.718} C_VEL
LIN {X 0,Y 528.048,Z 332.259,A -85,B 0,C 180,E1 -12218.208,E2 -12218.208} C_VEL
LIN {X 0,Y 528.086,Z 332.263,A -85,B 0,C 180,E1 -12220.634,E2 -12220.634} C_VEL
LIN {X 0,Y 528.058,Z 332.274,A -85,B 0,C 180,E1 -12221.766,E2 -12221.766} C_VEL
LIN {X 0,Y 532.797,Z 348.236,A -85,B 0,C 180,E1 -12222.165,E2 -12222.165} C_VEL
LIN {X 0,Y 531.333,Z 452.281,A -85,B 0,C 180,E1 -12223.854,E2 -12223.854} C_VEL
LIN {X 0,Y 531.178,Z 467.475,A -85,B 0,C 180,E1 -12224.268,E2 -12224.268} C_VEL
LIN {X 0,Y 530.885,Z 481.36,A -85,B 0,C 180,E1 -12224.797,E2 -12224.797} C_VEL
LIN {X 0,Y 530.5,Z 494.831,A -85,B 0,C 180,E1 -12225.471,E2 -12225.471} C_VEL
LIN {X 0,Y 530.035,Z 508.432,A -85,B 0,C 180,E1 -12226.336,E2 -12226.336} C_VEL
LIN {X 0,Y 529.555,Z 520.654,A -85,B 0,C 180,E1 -12227.297,E2 -12227.297} C_VEL
LIN {X 0,Y 529.113,Z 531.175,A -85,B 0,C 180,E1 -12228.3,E2 -12228.3} C_VEL
LIN {X 0,Y 528.745,Z 541.546,A -85,B 0,C 180,E1 -12229.505,E2 -12229.505} C_VEL
LIN {X 0,Y 528.35,Z 549.758,A -85,B 0,C 180,E1 -12230.653,E2 -12230.653} C_VEL
LIN {X 0,Y 527.973,Z 557.615,A -85,B 0,C 180,E1 -12231.992,E2 -12231.992} C_VEL
LIN {X 0,Y 527.763,Z 563.083,A -85,B 0,C 180,E1 -12233.14,E2 -12233.14} C_VEL
LIN {X 0,Y 527.527,Z 568.839,A -85,B 0,C 180,E1 -12234.667,E2 -12234.667} C_VEL
LIN {X 0,Y 527.499,Z 572.931,A -85,B 0,C 180,E1 -12236.193,E2 -12236.193} C_VEL
LIN {X 0,Y 527.459,Z 575.54,A -85,B 0,C 180,E1 -12237.717,E2 -12237.717} C_VEL
LIN {X 0,Y 527.396,Z 576.761,A -85,B 0,C 180,E1 -12239.239,E2 -12239.239} C_VEL
LIN {X 0,Y 527.411,Z 576.587,A -85,B 0,C 180,E1 -12240.761,E2 -12240.761} C_VEL
LIN {X 0,Y 527.682,Z 574.966,A -85,B 0,C 180,E1 -12242.282,E2 -12242.282} C_VEL
LIN {X 0,Y 528.198,Z 571.855,A -85,B 0,C 180,E1 -12243.802,E2 -12243.802} C_VEL
LIN {X 0,Y 528.448,Z 568.589,A -85,B 0,C 180,E1 -12244.942,E2 -12244.942} C_VEL
LIN {X 0,Y 528.619,Z 564.384,A -85,B 0,C 180,E1 -12246.085,E2 -12246.085} C_VEL
LIN {X 0,Y 529.369,Z 558.132,A -85,B 0,C 180,E1 -12247.412,E2 -12247.412} C_VEL
LIN {X 0,Y 529.959,Z 550.307,A -85,B 0,C 180,E1 -12248.742,E2 -12248.742} C_VEL
LIN {X 0,Y 530.562,Z 542.106,A -85,B 0,C 180,E1 -12249.882,E2 -12249.882} C_VEL
LIN {X 0,Y 531.224,Z 532.172,A -85,B 0,C 180,E1 -12251.022,E2 -12251.022} C_VEL
LIN {X 0,Y 531.814,Z 522.178,A -85,B 0,C 180,E1 -12251.972,E2 -12251.972} C_VEL
LIN {X 0,Y 532.61,Z 510.055,A -85,B 0,C 180,E1 -12252.919,E2 -12252.919} C_VEL
LIN {X 0,Y 533.268,Z 498.02,A -85,B 0,C 180,E1 -12253.676,E2 -12253.676} C_VEL
LIN {X 0,Y 533.683,Z 483.771,A -85,B 0,C 180,E1 -12254.392,E2 -12254.392} C_VEL
LIN {X 0,Y 534.04,Z 469.868,A -85,B 0,C 180,E1 -12254.916,E2 -12254.916} C_VEL
LIN {X 0,Y 534.256,Z 455.247,A -85,B 0,C 180,E1 -12255.299,E2 -12255.299} C_VEL
LIN {X 0,Y 536.268,Z 369.227,A -85,B 0,C 180,E1 -12256.839,E2 -12256.839} C_VEL
LIN {X 0,Y 536.739,Z 351.878,A -85,B 0,C 180,E1 -12257.164,E2 -12257.164} C_VEL
LIN {X 0,Y 530.617,Z 338.128,A -85,B 0,C 180,E1 -12257.785,E2 -12257.785} C_VEL
LIN {X 0,Y 528.224,Z 333.033,A -85,B 0,C 180,E1 -12258.036,E2 -12258.036} C_VEL
LIN {X 0,Y 528.094,Z 332.266,A -85,B 0,C 180,E1 -12258.08,E2 -12258.08} C_VEL
LIN {X 0,Y 528.081,Z 332.265,A -85,B 0,C 180,E1 -12260.985,E2 -12260.985} C_VEL
LIN {X 0,Y 528.052,Z 332.27,A -85,B 0,C 180,E1 -12263.756,E2 -12263.756} C_VEL
LIN {X 0,Y 528.043,Z 332.268,A -85,B 0,C 180,E1 -12266.808,E2 -12266.808} C_VEL
LIN {X 0,Y 528.064,Z 332.265,A -85,B 0,C 180,E1 -12269.392,E2 -12269.392} C_VEL
LIN {X 0,Y 528.036,Z 332.267,A -85,B 0,C 180,E1 -12272.046,E2 -12272.046} C_VEL
LIN {X 0,Y 528.058,Z 332.261,A -85,B 0,C 180,E1 -12274.776,E2 -12274.776} C_VEL
LIN {X 0,Y 528.055,Z 332.261,A -85,B 0,C 180,E1 -12277.261,E2 -12277.261} C_VEL
LIN {X 0,Y 528.013,Z 332.263,A -85,B 0,C 180,E1 -12280.543,E2 -12280.543} C_VEL
LIN {X 0,Y 528.03,Z 332.268,A -85,B 0,C 180,E1 -12283.148,E2 -12283.148} C_VEL
LIN {X 0,Y 528.036,Z 332.263,A -85,B 0,C 180,E1 -12285.751,E2 -12285.751} C_VEL
LIN {X 0,Y 528.019,Z 332.268,A -85,B 0,C 180,E1 -12288.449,E2 -12288.449} C_VEL
LIN {X 0,Y 527.992,Z 332.272,A -85,B 0,C 180,E1 -12291.427,E2 -12291.427} C_VEL
LIN {X 0,Y 528.017,Z 332.272,A -85,B 0,C 180,E1 -12294.29,E2 -12294.29} C_VEL
LIN {X 0,Y 527.983,Z 332.276,A -85,B 0,C 180,E1 -12297.049,E2 -12297.049} C_VEL
LIN {X 0,Y 528.081,Z 332.461,A -85,B 0,C 180,E1 -12299.843,E2 -12299.843} C_VEL
LIN {X 0,Y 532.045,Z 349.729,A -85,B 0,C 180,E1 -12302.253,E2 -12302.253} C_VEL
LIN {X 0,Y 533.232,Z 356.447,A -85,B 0,C 180,E1 -12303.151,E2 -12303.151} C_VEL
LIN {X 0,Y 532.106,Z 374.659,A -85,B 0,C 180,E1 -12305.369,E2 -12305.369} C_VEL
LIN {X 0,Y 530.699,Z 399.088,A -85,B 0,C 180,E1 -12308.311,E2 -12308.311} C_VEL
LIN {X 0,Y 529.599,Z 420.687,A -85,B 0,C 180,E1 -12310.892,E2 -12310.892} C_VEL
LIN {X 0,Y 529.466,Z 425.204,A -85,B 0,C 180,E1 -12311.4,E2 -12311.4} C_VEL
LIN {X 0,Y 530.942,Z 436.35,A -85,B 0,C 180,E1 -12311.668,E2 -12311.668} C_VEL
LIN {X 0,Y 534.133,Z 463.776,A -85,B 0,C 180,E1 -12312.171,E2 -12312.171} C_VEL
LIN {X 0,Y 534.436,Z 470.973,A -85,B 0,C 180,E1 -12312.282,E2 -12312.282} C_VEL
LIN {X 0,Y 533.356,Z 565.396,A -85,B 0,C 180,E1 -12313.576,E2 -12313.576} C_VEL
LIN {X 0,Y 532.75,Z 579.297,A -85,B 0,C 180,E1 -12313.904,E2 -12313.904} C_VEL
LIN {X 0,Y 531.967,Z 593.256,A -85,B 0,C 180,E1 -12314.389,E2 -12314.389} C_VEL
LIN {X 0,Y 531.081,Z 606.381,A -85,B 0,C 180,E1 -12314.999,E2 -12314.999} C_VEL
LIN {X 0,Y 530.207,Z 619.104,A -85,B 0,C 180,E1 -12315.756,E2 -12315.756} C_VEL
LIN {X 0,Y 529.328,Z 630.72,A -85,B 0,C 180,E1 -12316.61,E2 -12316.61} C_VEL
LIN {X 0,Y 528.817,Z 638.898,A -85,B 0,C 180,E1 -12317.279,E2 -12317.279} C_VEL
LIN {X 0,Y 528.303,Z 651.102,A -85,B 0,C 180,E1 -12318.238,E2 -12318.238} C_VEL
LIN {X 0,Y 527.814,Z 662.104,A -85,B 0,C 180,E1 -12319.293,E2 -12319.293} C_VEL
LIN {X 0,Y 527.433,Z 672.003,A -85,B 0,C 180,E1 -12320.444,E2 -12320.444} C_VEL
LIN {X 0,Y 527.053,Z 680.17,A -85,B 0,C 180,E1 -12321.594,E2 -12321.594} C_VEL
LIN {X 0,Y 526.861,Z 686.932,A -85,B 0,C 180,E1 -12322.744,E2 -12322.744} C_VEL
LIN {X 0,Y 526.724,Z 692.498,A -85,B 0,C 180,E1 -12323.893,E2 -12323.893} C_VEL
LIN {X 0,Y 526.66,Z 697.017,A -85,B 0,C 180,E1 -12325.041,E2 -12325.041} C_VEL
LIN {X 0,Y 526.588,Z 700.575,A -85,B 0,C 180,E1 -12326.186,E2 -12326.186} C_VEL
LIN {X 0,Y 526.578,Z 703.891,A -85,B 0,C 180,E1 -12327.713,E2 -12327.713} C_VEL
LIN {X 0,Y 526.53,Z 705.71,A -85,B 0,C 180,E1 -12329.238,E2 -12329.238} C_VEL
LIN {X 0,Y 526.529,Z 706.083,A -85,B 0,C 180,E1 -12330.762,E2 -12330.762} C_VEL
LIN {X 0,Y 526.581,Z 705.01,A -85,B 0,C 180,E1 -12332.287,E2 -12332.287} C_VEL
LIN {X 0,Y 526.587,Z 702.489,A -85,B 0,C 180,E1 -12333.813,E2 -12333.813} C_VEL
LIN {X 0,Y 526.745,Z 698.431,A -85,B 0,C 180,E1 -12335.341,E2 -12335.341} C_VEL
LIN {X 0,Y 526.893,Z 694.304,A -85,B 0,C 180,E1 -12336.488,E2 -12336.488} C_VEL
LIN {X 0,Y 527.094,Z 689.166,A -85,B 0,C 180,E1 -12337.636,E2 -12337.636} C_VEL
LIN {X 0,Y 527.489,Z 681.786,A -85,B 0,C 180,E1 -12338.976,E2 -12338.976} C_VEL
LIN {X 0,Y 528.035,Z 674.033,A -85,B 0,C 180,E1 -12340.123,E2 -12340.123} C_VEL
LIN {X 0,Y 528.557,Z 664.564,A -85,B 0,C 180,E1 -12341.29,E2 -12341.29} C_VEL
LIN {X 0,Y 529.238,Z 654.407,A -85,B 0,C 180,E1 -12342.322,E2 -12342.322} C_VEL
LIN {X 0,Y 529.942,Z 643.087,A -85,B 0,C 180,E1 -12343.277,E2 -12343.277} C_VEL
LIN {X 0,Y 530.737,Z 630.642,A -85,B 0,C 180,E1 -12344.132,E2 -12344.132} C_VEL
LIN {X 0,Y 531.451,Z 616.811,A -85,B 0,C 180,E1 -12344.892,E2 -12344.892} C_VEL
LIN {X 0,Y 532.083,Z 603.44,A -85,B 0,C 180,E1 -12345.46,E2 -12345.46} C_VEL
LIN {X 0,Y 532.654,Z 589.115,A -85,B 0,C 180,E1 -12345.908,E2 -12345.908} C_VEL
LIN {X 0,Y 533.157,Z 572.058,A -85,B 0,C 180,E1 -12346.252,E2 -12346.252} C_VEL
LIN {X 0,Y 535.446,Z 483.636,A -85,B 0,C 180,E1 -12347.854,E2 -12347.854} C_VEL
LIN {X 0,Y 535.78,Z 465.884,A -85,B 0,C 180,E1 -12348.2,E2 -12348.2} C_VEL
LIN {X 0,Y 534.096,Z 445.751,A -85,B 0,C 180,E1 -12348.711,E2 -12348.711} C_VEL
LIN {X 0,Y 532.647,Z 433.49,A -85,B 0,C 180,E1 -12349.079,E2 -12349.079} C_VEL
LIN {X 0,Y 530.013,Z 409.452,A -85,B 0,C 180,E1 -12350.142,E2 -12350.142} C_VEL
LIN {X 0,Y 529.66,Z 405.463,A -85,B 0,C 180,E1 -12350.338,E2 -12350.338} C_VEL
LIN {X 0,Y 530.72,Z 381.863,A -85,B 0,C 180,E1 -12353.119,E2 -12353.119} C_VEL
LIN {X 0,Y 532.04,Z 356.306,A -85,B 0,C 180,E1 -12356.153,E2 -12356.153} C_VEL
LIN {X 0,Y 532.118,Z 352.714,A -85,B 0,C 180,E1 -12356.587,E2 -12356.587} C_VEL
LIN {X 0,Y 528.841,Z 335.939,A -85,B 0,C 180,E1 -12358.773,E2 -12358.773} C_VEL
LIN {X 0,Y 528.076,Z 332.267,A -85,B 0,C 180,E1 -12359.263,E2 -12359.263} C_VEL
LIN {X 0,Y 527.999,Z 332.271,A -85,B 0,C 180,E1 -12362.049,E2 -12362.049} C_VEL
LIN {X 0,Y 527.993,Z 332.273,A -85,B 0,C 180,E1 -12364.781,E2 -12364.781} C_VEL
LIN {X 0,Y 527.976,Z 332.272,A -85,B 0,C 180,E1 -12367.609,E2 -12367.609} C_VEL
LIN {X 0,Y 528.008,Z 332.271,A -85,B 0,C 180,E1 -12370.543,E2 -12370.543} C_VEL
LIN {X 0,Y 528.041,Z 332.269,A -85,B 0,C 180,E1 -12373.613,E2 -12373.613} C_VEL
LIN {X 0,Y 528.041,Z 332.269,A -85,B 0,C 180,E1 -12376.388,E2 -12376.388} C_VEL
LIN {X 0,Y 528.009,Z 332.274,A -85,B 0,C 180,E1 -12379.457,E2 -12379.457} C_VEL
LIN {X 0,Y 528.046,Z 332.271,A -85,B 0,C 180,E1 -12382.739,E2 -12382.739} C_VEL
LIN {X 0,Y 528.023,Z 332.273,A -85,B 0,C 180,E1 -12385.332,E2 -12385.332} C_VEL
LIN {X 0,Y 528.037,Z 332.383,A -85,B 0,C 180,E1 -12388.023,E2 -12388.023} C_VEL
LIN {X 0,Y 532.826,Z 346.434,A -85,B 0,C 180,E1 -12390.184,E2 -12390.184} C_VEL
LIN {X 0,Y 535.531,Z 356.441,A -85,B 0,C 180,E1 -12391.603,E2 -12391.603} C_VEL
LIN {X 0,Y 536.927,Z 363.27,A -85,B 0,C 180,E1 -12392.51,E2 -12392.51} C_VEL
LIN {X 0,Y 535.514,Z 387.719,A -85,B 0,C 180,E1 -12395.257,E2 -12395.257} C_VEL
LIN {X 0,Y 533.946,Z 414.864,A -85,B 0,C 180,E1 -12398.248,E2 -12398.248} C_VEL
LIN {X 0,Y 532.76,Z 439.907,A -85,B 0,C 180,E1 -12401.001,E2 -12401.001} C_VEL
LIN {X 0,Y 535.644,Z 456.836,A -85,B 0,C 180,E1 -12401.511,E2 -12401.511} C_VEL
LIN {X 0,Y 536.535,Z 464.672,A -85,B 0,C 180,E1 -12401.716,E2 -12401.716} C_VEL
LIN {X 0,Y 534.164,Z 552.381,A -85,B 0,C 180,E1 -12403.307,E2 -12403.307} C_VEL
LIN {X 0,Y 533.336,Z 582.187,A -85,B 0,C 180,E1 -12403.849,E2 -12403.849} C_VEL
LIN {X 0,Y 532.764,Z 596.58,A -85,B 0,C 180,E1 -12404.267,E2 -12404.267} C_VEL
LIN {X 0,Y 532.045,Z 610.717,A -85,B 0,C 180,E1 -12404.832,E2 -12404.832} C_VEL
LIN {X 0,Y 531.265,Z 625.201,A -85,B 0,C 180,E1 -12405.59,E2 -12405.59} C_VEL
LIN {X 0,Y 530.417,Z 638.03,A -85,B 0,C 180,E1 -12406.444,E2 -12406.444} C_VEL
LIN {X 0,Y 529.617,Z 649.656,A -85,B 0,C 180,E1 -12407.396,E2 -12407.396} C_VEL
LIN {X 0,Y 528.825,Z 661.156,A -85,B 0,C 180,E1 -12408.54,E2 -12408.54} C_VEL
LIN {X 0,Y 528.267,Z 670.631,A -85,B 0,C 180,E1 -12409.689,E2 -12409.689} C_VEL
LIN {X 0,Y 527.596,Z 679.678,A -85,B 0,C 180,E1 -12411.026,E2 -12411.026} C_VEL
LIN {X 0,Y 527.17,Z 686.961,A -85,B 0,C 180,E1 -12412.365,E2 -12412.365} C_VEL
LIN {X 0,Y 526.924,Z 692.049,A -85,B 0,C 180,E1 -12413.512,E2 -12413.512} C_VEL
LIN {X 0,Y 526.656,Z 697.264,A -85,B 0,C 180,E1 -12415.041,E2 -12415.041} C_VEL
LIN {X 0,Y 526.588,Z 700.169,A -85,B 0,C 180,E1 -12416.187,E2 -12416.187} C_VEL
LIN {X 0,Y 526.511,Z 702.68,A -85,B 0,C 180,E1 -12417.713,E2 -12417.713} C_VEL
LIN {X 0,Y 526.462,Z 703.764,A -85,B 0,C 180,E1 -12419.238,E2 -12419.238} C_VEL
LIN {X 0,Y 526.461,Z 703.424,A -85,B 0,C 180,E1 -12420.763,E2 -12420.763} C_VEL
LIN {X 0,Y 526.508,Z 701.658,A -85,B 0,C 180,E1 -12422.288,E2 -12422.288} C_VEL
LIN {X 0,Y 526.524,Z 698.328,A -85,B 0,C 180,E1 -12423.853,E2 -12423.853} C_VEL
LIN {X 0,Y 526.646,Z 693.596,A -85,B 0,C 180,E1 -12425.342,E2 -12425.342} C_VEL
LIN {X 0,Y 526.75,Z 688.883,A -85,B 0,C 180,E1 -12426.49,E2 -12426.49} C_VEL
LIN {X 0,Y 527.025,Z 681.984,A -85,B 0,C 180,E1 -12427.83,E2 -12427.83} C_VEL
LIN {X 0,Y 527.372,Z 673.388,A -85,B 0,C 180,E1 -12429.171,E2 -12429.171} C_VEL
LIN {X 0,Y 527.828,Z 664.406,A -85,B 0,C 180,E1 -12430.32,E2 -12430.32} C_VEL
LIN {X 0,Y 528.303,Z 653.536,A -85,B 0,C 180,E1 -12431.471,E2 -12431.471} C_VEL
LIN {X 0,Y 528.773,Z 642.537,A -85,B 0,C 180,E1 -12432.431,E2 -12432.431} C_VEL
LIN {X 0,Y 529.37,Z 630.501,A -85,B 0,C 180,E1 -12433.291,E2 -12433.291} C_VEL
LIN {X 0,Y 529.993,Z 617.25,A -85,B 0,C 180,E1 -12434.055,E2 -12434.055} C_VEL
LIN {X 0,Y 530.494,Z 603.5,A -85,B 0,C 180,E1 -12434.676,E2 -12434.676} C_VEL
LIN {X 0,Y 530.879,Z 588.521,A -85,B 0,C 180,E1 -12435.178,E2 -12435.178} C_VEL
LIN {X 0,Y 531.291,Z 573.374,A -85,B 0,C 180,E1 -12435.508,E2 -12435.508} C_VEL
LIN {X 0,Y 532.951,Z 461.445,A -85,B 0,C 180,E1 -12437.327,E2 -12437.327} C_VEL
LIN {X 0,Y 530.403,Z 439.589,A -85,B 0,C 180,E1 -12437.772,E2 -12437.772} C_VEL
LIN {X 0,Y 531.566,Z 407.871,A -85,B 0,C 180,E1 -12441.246,E2 -12441.246} C_VEL
LIN {X 0,Y 532.758,Z 380.453,A -85,B 0,C 180,E1 -12444.259,E2 -12444.259} C_VEL
LIN {X 0,Y 533.648,Z 357.367,A -85,B 0,C 180,E1 -12446.806,E2 -12446.806} C_VEL
LIN {X 0,Y 529.379,Z 337.971,A -85,B 0,C 180,E1 -12449.158,E2 -12449.158} C_VEL
LIN {X 0,Y 528.069,Z 332.266,A -85,B 0,C 180,E1 -12449.884,E2 -12449.884} C_VEL
LIN {X 0,Y 528.04,Z 332.269,A -85,B 0,C 180,E1 -12452.947,E2 -12452.947} C_VEL
LIN {X 0,Y 528.108,Z 332.255,A -85,B 0,C 180,E1 -12455.996,E2 -12455.996} C_VEL
LIN {X 0,Y 528.006,Z 332.269,A -85,B 0,C 180,E1 -12458.572,E2 -12458.572} C_VEL
LIN {X 0,Y 528.07,Z 332.265,A -85,B 0,C 180,E1 -12460.882,E2 -12460.882} C_VEL
LIN {X 0,Y 528.057,Z 332.262,A -85,B 0,C 180,E1 -12463.611,E2 -12463.611} C_VEL
LIN {X 0,Y 528.057,Z 332.263,A -85,B 0,C 180,E1 -12466.389,E2 -12466.389} C_VEL
LIN {X 0,Y 528.083,Z 332.259,A -85,B 0,C 180,E1 -12469.464,E2 -12469.464} C_VEL
LIN {X 0,Y 528.056,Z 332.269,A -85,B 0,C 180,E1 -12472.739,E2 -12472.739} C_VEL
LIN {X 0,Y 528.058,Z 332.262,A -85,B 0,C 180,E1 -12475.327,E2 -12475.327} C_VEL
LIN {X 0,Y 528.041,Z 332.266,A -85,B 0,C 180,E1 -12478.099,E2 -12478.099} C_VEL
LIN {X 0,Y 528.056,Z 332.263,A -85,B 0,C 180,E1 -12481.101,E2 -12481.101} C_VEL
LIN {X 0,Y 528.047,Z 332.267,A -85,B 0,C 180,E1 -12484.04,E2 -12484.04} C_VEL
LIN {X 0,Y 528.05,Z 332.267,A -85,B 0,C 180,E1 -12486.55,E2 -12486.55} C_VEL
LIN {X 0,Y 528.081,Z 332.259,A -85,B 0,C 180,E1 -12489.015,E2 -12489.015} C_VEL
LIN {X 0,Y 528.057,Z 332.262,A -85,B 0,C 180,E1 -12491.437,E2 -12491.437} C_VEL
LIN {X 0,Y 528.076,Z 332.265,A -85,B 0,C 180,E1 -12493.827,E2 -12493.827} C_VEL
LIN {X 0,Y 528.132,Z 332.257,A -85,B 0,C 180,E1 -12496.189,E2 -12496.189} C_VEL
LIN {X 0,Y 528.097,Z 332.26,A -85,B 0,C 180,E1 -12497.381,E2 -12497.381} C_VEL
LIN {X 0,Y 533.843,Z 349.414,A -85,B 0,C 180,E1 -12497.804,E2 -12497.804} C_VEL
LIN {X 0,Y 533.683,Z 362.577,A -85,B 0,C 180,E1 -12497.98,E2 -12497.98} C_VEL
LIN {X 0,Y 532.941,Z 368.415,A -85,B 0,C 180,E1 -12498.037,E2 -12498.037} C_VEL
LIN {X 0,Y 527.304,Z 387.402,A -85,B 0,C 180,E1 -12498.126,E2 -12498.126} C_VEL
LIN {X 0,Y 526.586,Z 393.24,A -85,B 0,C 180,E1 -12498.185,E2 -12498.185} C_VEL
LIN {X 0,Y 526.095,Z 453.1,A -85,B 0,C 180,E1 -12499.015,E2 -12499.015} C_VEL
LIN {X 0,Y 525.972,Z 467.409,A -85,B 0,C 180,E1 -12499.352,E2 -12499.352} C_VEL
LIN {X 0,Y 525.705,Z 481.068,A -85,B 0,C 180,E1 -12499.832,E2 -12499.832} C_VEL
LIN {X 0,Y 525.294,Z 493.397,A -85,B 0,C 180,E1 -12500.405,E2 -12500.405} C_VEL
LIN {X 0,Y 524.768,Z 506.323,A -85,B 0,C 180,E1 -12501.176,E2 -12501.176} C_VEL
LIN {X 0,Y 524.248,Z 517.872,A -85,B 0,C 180,E1 -12502.032,E2 -12502.032} C_VEL
LIN {X 0,Y 523.495,Z 529.487,A -85,B 0,C 180,E1 -12503.084,E2 -12503.084} C_VEL
LIN {X 0,Y 522.753,Z 539.863,A -85,B 0,C 180,E1 -12504.233,E2 -12504.233} C_VEL
LIN {X 0,Y 522.183,Z 548.421,A -85,B 0,C 180,E1 -12505.384,E2 -12505.384} C_VEL
LIN {X 0,Y 521.691,Z 556.627,A -85,B 0,C 180,E1 -12506.729,E2 -12506.729} C_VEL
LIN {X 0,Y 521.23,Z 563.25,A -85,B 0,C 180,E1 -12508.075,E2 -12508.075} C_VEL
LIN {X 0,Y 520.852,Z 567.815,A -85,B 0,C 180,E1 -12509.23,E2 -12509.23} C_VEL
LIN {X 0,Y 520.548,Z 572.55,A -85,B 0,C 180,E1 -12510.771,E2 -12510.771} C_VEL
LIN {X 0,Y 520.511,Z 575.824,A -85,B 0,C 180,E1 -12512.314,E2 -12512.314} C_VEL
LIN {X 0,Y 520.437,Z 577.766,A -85,B 0,C 180,E1 -12513.859,E2 -12513.859} C_VEL
LIN {X 0,Y 520.478,Z 578.398,A -85,B 0,C 180,E1 -12515.406,E2 -12515.406} C_VEL
LIN {X 0,Y 520.561,Z 577.737,A -85,B 0,C 180,E1 -12516.956,E2 -12516.956} C_VEL
LIN {X 0,Y 520.726,Z 575.766,A -85,B 0,C 180,E1 -12518.509,E2 -12518.509} C_VEL
LIN {X 0,Y 521.132,Z 572.41,A -85,B 0,C 180,E1 -12520.063,E2 -12520.063} C_VEL
LIN {X 0,Y 521.555,Z 567.583,A -85,B 0,C 180,E1 -12521.622,E2 -12521.622} C_VEL
LIN {X 0,Y 522.182,Z 561.115,A -85,B 0,C 180,E1 -12523.182,E2 -12523.182} C_VEL
LIN {X 0,Y 522.819,Z 553.886,A -85,B 0,C 180,E1 -12524.549,E2 -12524.549} C_VEL
LIN {X 0,Y 523.666,Z 544.839,A -85,B 0,C 180,E1 -12525.915,E2 -12525.915} C_VEL
LIN {X 0,Y 524.446,Z 535.343,A -85,B 0,C 180,E1 -12527.088,E2 -12527.088} C_VEL
LIN {X 0,Y 525.216,Z 524.772,A -85,B 0,C 180,E1 -12528.164,E2 -12528.164} C_VEL
LIN {X 0,Y 525.886,Z 514.141,A -85,B 0,C 180,E1 -12529.06,E2 -12529.06} C_VEL
LIN {X 0,Y 526.657,Z 501.462,A -85,B 0,C 180,E1 -12529.926,E2 -12529.926} C_VEL
LIN {X 0,Y 527.278,Z 487.815,A -85,B 0,C 180,E1 -12530.663,E2 -12530.663} C_VEL
LIN {X 0,Y 527.628,Z 474.679,A -85,B 0,C 180,E1 -12531.204,E2 -12531.204} C_VEL
LIN {X 0,Y 527.84,Z 460.596,A -85,B 0,C 180,E1 -12531.619,E2 -12531.619} C_VEL
LIN {X 0,Y 528.017,Z 446.125,A -85,B 0,C 180,E1 -12531.881,E2 -12531.881} C_VEL
LIN {X 0,Y 529.022,Z 353.242,A -85,B 0,C 180,E1 -12533.158,E2 -12533.158} C_VEL
LIN {X 0,Y 521.062,Z 333.54,A -85,B 0,C 180,E1 -12533.774,E2 -12533.774} C_VEL
LIN {X 0,Y 521.004,Z 333.151,A -85,B 0,C 180,E1 -12533.786,E2 -12533.786} C_VEL
LIN {X 0,Y 521.002,Z 333.148,A -85,B 0,C 180,E1 -12536.338,E2 -12536.338} C_VEL
LIN {X 0,Y 521.013,Z 333.143,A -85,B 0,C 180,E1 -12539.09,E2 -12539.09} C_VEL
LIN {X 0,Y 520.953,Z 333.153,A -85,B 0,C 180,E1 -12542.106,E2 -12542.106} C_VEL
LIN {X 0,Y 520.959,Z 333.147,A -85,B 0,C 180,E1 -12545.321,E2 -12545.321} C_VEL
LIN {X 0,Y 520.942,Z 333.155,A -85,B 0,C 180,E1 -12548.207,E2 -12548.207} C_VEL
LIN {X 0,Y 520.973,Z 333.147,A -85,B 0,C 180,E1 -12551.209,E2 -12551.209} C_VEL
LIN {X 0,Y 520.99,Z 333.143,A -85,B 0,C 180,E1 -12554.556,E2 -12554.556} C_VEL
LIN {X 0,Y 521.005,Z 333.144,A -85,B 0,C 180,E1 -12557.762,E2 -12557.762} C_VEL
LIN {X 0,Y 520.937,Z 333.145,A -85,B 0,C 180,E1 -12560.805,E2 -12560.805} C_VEL
LIN {X 0,Y 520.976,Z 333.123,A -85,B 0,C 180,E1 -12563.774,E2 -12563.774} C_VEL
LIN {X 0,Y 520.98,Z 333.142,A -85,B 0,C 180,E1 -12566.548,E2 -12566.548} C_VEL
LIN {X 0,Y 520.995,Z 333.139,A -85,B 0,C 180,E1 -12569.367,E2 -12569.367} C_VEL
LIN {X 0,Y 520.978,Z 333.148,A -85,B 0,C 180,E1 -12571.929,E2 -12571.929} C_VEL
LIN {X 0,Y 520.986,Z 333.138,A -85,B 0,C 180,E1 -12574.518,E2 -12574.518} C_VEL
LIN {X 0,Y 520.969,Z 333.146,A -85,B 0,C 180,E1 -12577.051,E2 -12577.051} C_VEL
LIN {X 0,Y 521.034,Z 333.142,A -85,B 0,C 180,E1 -12580.361,E2 -12580.361} C_VEL
LIN {X 0,Y 521.016,Z 333.152,A -85,B 0,C 180,E1 -12581.601,E2 -12581.601} C_VEL
LIN {X 0,Y 525.88,Z 349.206,A -85,B 0,C 180,E1 -12582.007,E2 -12582.007} C_VEL
LIN {X 0,Y 524.346,Z 452.871,A -85,B 0,C 180,E1 -12583.728,E2 -12583.728} C_VEL
LIN {X 0,Y 524.184,Z 468.446,A -85,B 0,C 180,E1 -12584.159,E2 -12584.159} C_VEL
LIN {X 0,Y 523.879,Z 482.085,A -85,B 0,C 180,E1 -12584.688,E2 -12584.688} C_VEL
LIN {X 0,Y 523.486,Z 495.552,A -85,B 0,C 180,E1 -12585.371,E2 -12585.371} C_VEL
LIN {X 0,Y 523.019,Z 509.159,A -85,B 0,C 180,E1 -12586.248,E2 -12586.248} C_VEL
LIN {X 0,Y 522.537,Z 521.397,A -85,B 0,C 180,E1 -12587.222,E2 -12587.222} C_VEL
LIN {X 0,Y 522.105,Z 531.7,A -85,B 0,C 180,E1 -12588.214,E2 -12588.214} C_VEL
LIN {X 0,Y 521.763,Z 541.577,A -85,B 0,C 180,E1 -12589.363,E2 -12589.363} C_VEL
LIN {X 0,Y 521.314,Z 549.926,A -85,B 0,C 180,E1 -12590.526,E2 -12590.526} C_VEL
LIN {X 0,Y 520.931,Z 557.908,A -85,B 0,C 180,E1 -12591.883,E2 -12591.883} C_VEL
LIN {X 0,Y 520.713,Z 563.484,A -85,B 0,C 180,E1 -12593.046,E2 -12593.046} C_VEL
LIN {X 0,Y 520.484,Z 569.344,A -85,B 0,C 180,E1 -12594.594,E2 -12594.594} C_VEL
LIN {X 0,Y 520.435,Z 573.568,A -85,B 0,C 180,E1 -12596.141,E2 -12596.141} C_VEL
LIN {X 0,Y 520.5,Z 575.084,A -85,B 0,C 180,E1 -12596.914,E2 -12596.914} C_VEL
LIN {X 0,Y 520.359,Z 577.084,A -85,B 0,C 180,E1 -12598.457,E2 -12598.457} C_VEL
LIN {X 0,Y 520.341,Z 577.686,A -85,B 0,C 180,E1 -12600,E2 -12600} C_VEL
LIN {X 0,Y 520.484,Z 576.882,A -85,B 0,C 180,E1 -12601.542,E2 -12601.542} C_VEL
LIN {X 0,Y 520.921,Z 574.61,A -85,B 0,C 180,E1 -12603.083,E2 -12603.083} C_VEL
LIN {X 0,Y 521.44,Z 570.827,A -85,B 0,C 180,E1 -12604.623,E2 -12604.623} C_VEL
LIN {X 0,Y 521.675,Z 565.543,A -85,B 0,C 180,E1 -12606.166,E2 -12606.166} C_VEL
LIN {X 0,Y 522.307,Z 560.338,A -85,B 0,C 180,E1 -12607.319,E2 -12607.319} C_VEL
LIN {X 0,Y 522.986,Z 552.873,A -85,B 0,C 180,E1 -12608.666,E2 -12608.666} C_VEL
LIN {X 0,Y 523.592,Z 545.027,A -85,B 0,C 180,E1 -12609.821,E2 -12609.821} C_VEL
LIN {X 0,Y 524.302,Z 535.542,A -85,B 0,C 180,E1 -12610.974,E2 -12610.974} C_VEL
LIN {X 0,Y 524.952,Z 524.979,A -85,B 0,C 180,E1 -12612.033,E2 -12612.033} C_VEL
LIN {X 0,Y 525.757,Z 513.242,A -85,B 0,C 180,E1 -12612.992,E2 -12612.992} C_VEL
LIN {X 0,Y 526.566,Z 500.216,A -85,B 0,C 180,E1 -12613.853,E2 -12613.853} C_VEL
LIN {X 0,Y 527.055,Z 486.352,A -85,B 0,C 180,E1 -12614.577,E2 -12614.577} C_VEL
LIN {X 0,Y 527.434,Z 472.36,A -85,B 0,C 180,E1 -12615.132,E2 -12615.132} C_VEL
LIN {X 0,Y 527.654,Z 457.738,A -85,B 0,C 180,E1 -12615.544,E2 -12615.544} C_VEL
LIN {X 0,Y 529.668,Z 376.316,A -85,B 0,C 180,E1 -12617.041,E2 -12617.041} C_VEL
LIN {X 0,Y 530.28,Z 353.638,A -85,B 0,C 180,E1 -12617.477,E2 -12617.477} C_VEL
LIN {X 0,Y 523.893,Z 339.492,A -85,B 0,C 180,E1 -12618.153,E2 -12618.153} C_VEL
LIN {X 0,Y 521.18,Z 333.955,A -85,B 0,C 180,E1 -12618.439,E2 -12618.439} C_VEL
LIN {X 0,Y 521.036,Z 333.145,A -85,B 0,C 180,E1 -12618.502,E2 -12618.502} C_VEL
LIN {X 0,Y 521.025,Z 333.144,A -85,B 0,C 180,E1 -12621.283,E2 -12621.283} C_VEL
LIN {X 0,Y 521.026,Z 333.146,A -85,B 0,C 180,E1 -12623.912,E2 -12623.912} C_VEL
LIN {X 0,Y 521.02,Z 333.144,A -85,B 0,C 180,E1 -12627.199,E2 -12627.199} C_VEL
LIN {X 0,Y 521.021,Z 333.145,A -85,B 0,C 180,E1 -12629.829,E2 -12629.829} C_VEL
LIN {X 0,Y 520.976,Z 333.145,A -85,B 0,C 180,E1 -12632.533,E2 -12632.533} C_VEL
LIN {X 0,Y 521.015,Z 333.139,A -85,B 0,C 180,E1 -12635.316,E2 -12635.316} C_VEL
LIN {X 0,Y 521.021,Z 333.138,A -85,B 0,C 180,E1 -12637.516,E2 -12637.516} C_VEL
LIN {X 0,Y 520.965,Z 333.141,A -85,B 0,C 180,E1 -12640.193,E2 -12640.193} C_VEL
LIN {X 0,Y 520.989,Z 333.146,A -85,B 0,C 180,E1 -12643.288,E2 -12643.288} C_VEL
LIN {X 0,Y 520.996,Z 333.142,A -85,B 0,C 180,E1 -12646.552,E2 -12646.552} C_VEL
LIN {X 0,Y 520.975,Z 333.151,A -85,B 0,C 180,E1 -12648.843,E2 -12648.843} C_VEL
LIN {X 0,Y 520.933,Z 333.151,A -85,B 0,C 180,E1 -12651.792,E2 -12651.792} C_VEL
LIN {X 0,Y 520.954,Z 333.148,A -85,B 0,C 180,E1 -12654.679,E2 -12654.679} C_VEL
LIN {X 0,Y 520.95,Z 333.152,A -85,B 0,C 180,E1 -12657.894,E2 -12657.894} C_VEL
LIN {X 0,Y 521.039,Z 333.247,A -85,B 0,C 180,E1 -12659.573,E2 -12659.573} C_VEL
LIN {X 0,Y 524.886,Z 349.952,A -85,B 0,C 180,E1 -12661.945,E2 -12661.945} C_VEL
LIN {X 0,Y 526.381,Z 358.445,A -85,B 0,C 180,E1 -12663.1,E2 -12663.1} C_VEL
LIN {X 0,Y 525.131,Z 377.405,A -85,B 0,C 180,E1 -12665.437,E2 -12665.437} C_VEL
LIN {X 0,Y 523.592,Z 403.506,A -85,B 0,C 180,E1 -12668.62,E2 -12668.62} C_VEL
LIN {X 0,Y 522.544,Z 423.001,A -85,B 0,C 180,E1 -12670.98,E2 -12670.98} C_VEL
LIN {X 0,Y 524.871,Z 441.595,A -85,B 0,C 180,E1 -12671.508,E2 -12671.508} C_VEL
LIN {X 0,Y 527.744,Z 468.127,A -85,B 0,C 180,E1 -12671.995,E2 -12671.995} C_VEL
LIN {X 0,Y 526.579,Z 564.557,A -85,B 0,C 180,E1 -12673.332,E2 -12673.332} C_VEL
LIN {X 0,Y 525.981,Z 578.737,A -85,B 0,C 180,E1 -12673.674,E2 -12673.674} C_VEL
LIN {X 0,Y 525.192,Z 591.91,A -85,B 0,C 180,E1 -12674.133,E2 -12674.133} C_VEL
LIN {X 0,Y 524.365,Z 604.272,A -85,B 0,C 180,E1 -12674.703,E2 -12674.703} C_VEL
LIN {X 0,Y 523.405,Z 617.245,A -85,B 0,C 180,E1 -12675.468,E2 -12675.468} C_VEL
LIN {X 0,Y 522.389,Z 630.228,A -85,B 0,C 180,E1 -12676.429,E2 -12676.429} C_VEL
LIN {X 0,Y 521.673,Z 640.42,A -85,B 0,C 180,E1 -12677.299,E2 -12677.299} C_VEL
LIN {X 0,Y 521.208,Z 652.379,A -85,B 0,C 180,E1 -12678.272,E2 -12678.272} C_VEL
LIN {X 0,Y 520.702,Z 663.178,A -85,B 0,C 180,E1 -12679.341,E2 -12679.341} C_VEL
LIN {X 0,Y 520.345,Z 672.913,A -85,B 0,C 180,E1 -12680.508,E2 -12680.508} C_VEL
LIN {X 0,Y 519.965,Z 680.932,A -85,B 0,C 180,E1 -12681.673,E2 -12681.673} C_VEL
LIN {X 0,Y 519.743,Z 688.55,A -85,B 0,C 180,E1 -12683.033,E2 -12683.033} C_VEL
LIN {X 0,Y 519.64,Z 693.846,A -85,B 0,C 180,E1 -12684.198,E2 -12684.198} C_VEL
LIN {X 0,Y 519.519,Z 698.06,A -85,B 0,C 180,E1 -12685.36,E2 -12685.36} C_VEL
LIN {X 0,Y 519.511,Z 700.368,A -85,B 0,C 180,E1 -12686.134,E2 -12686.134} C_VEL
LIN {X 0,Y 519.492,Z 703.777,A -85,B 0,C 180,E1 -12687.682,E2 -12687.682} C_VEL
LIN {X 0,Y 519.456,Z 705.654,A -85,B 0,C 180,E1 -12689.227,E2 -12689.227} C_VEL
LIN {X 0,Y 519.455,Z 706.08,A -85,B 0,C 180,E1 -12690.772,E2 -12690.772} C_VEL
LIN {X 0,Y 519.496,Z 705.059,A -85,B 0,C 180,E1 -12692.318,E2 -12692.318} C_VEL
LIN {X 0,Y 519.511,Z 702.585,A -85,B 0,C 180,E1 -12693.865,E2 -12693.865} C_VEL
LIN {X 0,Y 519.664,Z 698.592,A -85,B 0,C 180,E1 -12695.414,E2 -12695.414} C_VEL
LIN {X 0,Y 519.85,Z 694.497,A -85,B 0,C 180,E1 -12696.576,E2 -12696.576} C_VEL
LIN {X 0,Y 520.063,Z 689.42,A -85,B 0,C 180,E1 -12697.74,E2 -12697.74} C_VEL
LIN {X 0,Y 520.485,Z 682.094,A -85,B 0,C 180,E1 -12699.098,E2 -12699.098} C_VEL
LIN {X 0,Y 521.041,Z 674.396,A -85,B 0,C 180,E1 -12700.26,E2 -12700.26} C_VEL
LIN {X 0,Y 521.639,Z 664.752,A -85,B 0,C 180,E1 -12701.473,E2 -12701.473} C_VEL
LIN {X 0,Y 522.426,Z 653.957,A -85,B 0,C 180,E1 -12702.584,E2 -12702.584} C_VEL
LIN {X 0,Y 523.148,Z 642.535,A -85,B 0,C 180,E1 -12703.551,E2 -12703.551} C_VEL
LIN {X 0,Y 524.005,Z 630.006,A -85,B 0,C 180,E1 -12704.416,E2 -12704.416} C_VEL
LIN {X 0,Y 524.781,Z 616.095,A -85,B 0,C 180,E1 -12705.185,E2 -12705.185} C_VEL
LIN {X 0,Y 525.472,Z 602.588,A -85,B 0,C 180,E1 -12705.759,E2 -12705.759} C_VEL
LIN {X 0,Y 526.028,Z 588.816,A -85,B 0,C 180,E1 -12706.188,E2 -12706.188} C_VEL
LIN {X 0,Y 526.635,Z 569.773,A -85,B 0,C 180,E1 -12706.573,E2 -12706.573} C_VEL
LIN {X 0,Y 529.118,Z 481.301,A -85,B 0,C 180,E1 -12708.225,E2 -12708.225} C_VEL
LIN {X 0,Y 529.382,Z 466.894,A -85,B 0,C 180,E1 -12708.515,E2 -12708.515} C_VEL
LIN {X 0,Y 527.821,Z 447.285,A -85,B 0,C 180,E1 -12709.024,E2 -12709.024} C_VEL
LIN {X 0,Y 526.273,Z 434.434,A -85,B 0,C 180,E1 -12709.418,E2 -12709.418} C_VEL
LIN {X 0,Y 523.908,Z 411.263,A -85,B 0,C 180,E1 -12710.479,E2 -12710.479} C_VEL
LIN {X 0,Y 522.849,Z 401.453,A -85,B 0,C 180,E1 -12710.979,E2 -12710.979} C_VEL
LIN {X 0,Y 523.917,Z 379.143,A -85,B 0,C 180,E1 -12713.646,E2 -12713.646} C_VEL
LIN {X 0,Y 525.175,Z 355.997,A -85,B 0,C 180,E1 -12716.433,E2 -12716.433} C_VEL
LIN {X 0,Y 524.799,Z 351.612,A -85,B 0,C 180,E1 -12716.987,E2 -12716.987} C_VEL
LIN {X 0,Y 521.044,Z 333.142,A -85,B 0,C 180,E1 -12719.469,E2 -12719.469} C_VEL
LIN {X 0,Y 520.931,Z 333.151,A -85,B 0,C 180,E1 -12722.537,E2 -12722.537} C_VEL
LIN {X 0,Y 520.952,Z 333.15,A -85,B 0,C 180,E1 -12725.321,E2 -12725.321} C_VEL
LIN {X 0,Y 520.925,Z 333.152,A -85,B 0,C 180,E1 -12728.208,E2 -12728.208} C_VEL
LIN {X 0,Y 520.969,Z 333.146,A -85,B 0,C 180,E1 -12731.209,E2 -12731.209} C_VEL
LIN {X 0,Y 520.985,Z 333.149,A -85,B 0,C 180,E1 -12734.556,E2 -12734.556} C_VEL
LIN {X 0,Y 520.958,Z 333.151,A -85,B 0,C 180,E1 -12737.758,E2 -12737.758} C_VEL
LIN {X 0,Y 520.936,Z 333.153,A -85,B 0,C 180,E1 -12740.805,E2 -12740.805} C_VEL
LIN {X 0,Y 521.03,Z 333.142,A -85,B 0,C 180,E1 -12743.766,E2 -12743.766} C_VEL
LIN {X 0,Y 520.985,Z 333.151,A -85,B 0,C 180,E1 -12747.009,E2 -12747.009} C_VEL
LIN {X 0,Y 520.983,Z 333.315,A -85,B 0,C 180,E1 -12747.41,E2 -12747.41} C_VEL
LIN {X 0,Y 525.293,Z 345.413,A -85,B 0,C 180,E1 -12749.38,E2 -12749.38} C_VEL
LIN {X 0,Y 528.54,Z 356.312,A -85,B 0,C 180,E1 -12751.005,E2 -12751.005} C_VEL
LIN {X 0,Y 530.526,Z 366.152,A -85,B 0,C 180,E1 -12752.352,E2 -12752.352} C_VEL
LIN {X 0,Y 528.858,Z 392.537,A -85,B 0,C 180,E1 -12755.342,E2 -12755.342} C_VEL
LIN {X 0,Y 527.234,Z 419.012,A -85,B 0,C 180,E1 -12758.31,E2 -12758.31} C_VEL
LIN {X 0,Y 526.139,Z 439.647,A -85,B 0,C 180,E1 -12760.616,E2 -12760.616} C_VEL
LIN {X 0,Y 529.032,Z 456.282,A -85,B 0,C 180,E1 -12761.144,E2 -12761.144} C_VEL
LIN {X 0,Y 530.109,Z 465.953,A -85,B 0,C 180,E1 -12761.405,E2 -12761.405} C_VEL
LIN {X 0,Y 527.633,Z 550.169,A -85,B 0,C 180,E1 -12762.974,E2 -12762.974} C_VEL
LIN {X 0,Y 526.705,Z 582.426,A -85,B 0,C 180,E1 -12763.579,E2 -12763.579} C_VEL
LIN {X 0,Y 526.087,Z 597.009,A -85,B 0,C 180,E1 -12764.012,E2 -12764.012} C_VEL
LIN {X 0,Y 525.389,Z 609.987,A -85,B 0,C 180,E1 -12764.536,E2 -12764.536} C_VEL
LIN {X 0,Y 524.702,Z 622.897,A -85,B 0,C 180,E1 -12765.208,E2 -12765.208} C_VEL
LIN {X 0,Y 523.863,Z 634.83,A -85,B 0,C 180,E1 -12765.975,E2 -12765.975} C_VEL
LIN {X 0,Y 522.952,Z 647.087,A -85,B 0,C 180,E1 -12766.937,E2 -12766.937} C_VEL
LIN {X 0,Y 522.193,Z 658.152,A -85,B 0,C 180,E1 -12768,E2 -12768} C_VEL
LIN {X 0,Y 521.561,Z 668.096,A -85,B 0,C 180,E1 -12769.163,E2 -12769.163} C_VEL
LIN {X 0,Y 520.813,Z 677.629,A -85,B 0,C 180,E1 -12770.517,E2 -12770.517} C_VEL
LIN {X 0,Y 520.294,Z 685.353,A -85,B 0,C 180,E1 -12771.874,E2 -12771.874} C_VEL
LIN {X 0,Y 519.967,Z 690.703,A -85,B 0,C 180,E1 -12773.037,E2 -12773.037} C_VEL
LIN {X 0,Y 519.617,Z 696.327,A -85,B 0,C 180,E1 -12774.586,E2 -12774.586} C_VEL
LIN {X 0,Y 519.512,Z 700.298,A -85,B 0,C 180,E1 -12776.135,E2 -12776.135} C_VEL
LIN {X 0,Y 519.43,Z 702.762,A -85,B 0,C 180,E1 -12777.682,E2 -12777.682} C_VEL
LIN {X 0,Y 519.391,Z 703.794,A -85,B 0,C 180,E1 -12779.227,E2 -12779.227} C_VEL
LIN {X 0,Y 519.39,Z 703.4,A -85,B 0,C 180,E1 -12780.773,E2 -12780.773} C_VEL
LIN {X 0,Y 519.407,Z 701.576,A -85,B 0,C 180,E1 -12782.319,E2 -12782.319} C_VEL
LIN {X 0,Y 519.434,Z 698.265,A -85,B 0,C 180,E1 -12783.866,E2 -12783.866} C_VEL
LIN {X 0,Y 519.563,Z 693.345,A -85,B 0,C 180,E1 -12785.415,E2 -12785.415} C_VEL
LIN {X 0,Y 519.676,Z 688.555,A -85,B 0,C 180,E1 -12786.579,E2 -12786.579} C_VEL
LIN {X 0,Y 519.951,Z 681.56,A -85,B 0,C 180,E1 -12787.937,E2 -12787.937} C_VEL
LIN {X 0,Y 520.344,Z 672.859,A -85,B 0,C 180,E1 -12789.296,E2 -12789.296} C_VEL
LIN {X 0,Y 520.791,Z 663.755,A -85,B 0,C 180,E1 -12790.461,E2 -12790.461} C_VEL
LIN {X 0,Y 521.275,Z 652.729,A -85,B 0,C 180,E1 -12791.628,E2 -12791.628} C_VEL
LIN {X 0,Y 521.83,Z 641.516,A -85,B 0,C 180,E1 -12792.599,E2 -12792.599} C_VEL
LIN {X 0,Y 522.44,Z 629.246,A -85,B 0,C 180,E1 -12793.471,E2 -12793.471} C_VEL
LIN {X 0,Y 523.024,Z 615.691,A -85,B 0,C 180,E1 -12794.246,E2 -12794.246} C_VEL
LIN {X 0,Y 523.598,Z 601.542,A -85,B 0,C 180,E1 -12794.873,E2 -12794.873} C_VEL
LIN {X 0,Y 523.956,Z 587.356,A -85,B 0,C 180,E1 -12795.334,E2 -12795.334} C_VEL
LIN {X 0,Y 524.319,Z 572.068,A -85,B 0,C 180,E1 -12795.663,E2 -12795.663} C_VEL
LIN {X 0,Y 526.082,Z 462.323,A -85,B 0,C 180,E1 -12797.487,E2 -12797.487} C_VEL
LIN {X 0,Y 523.397,Z 439.577,A -85,B 0,C 180,E1 -12797.959,E2 -12797.959} C_VEL
LIN {X 0,Y 524.601,Z 408.981,A -85,B 0,C 180,E1 -12801.337,E2 -12801.337} C_VEL
LIN {X 0,Y 525.727,Z 383.259,A -85,B 0,C 180,E1 -12804.186,E2 -12804.186} C_VEL
LIN {X 0,Y 526.759,Z 359.053,A -85,B 0,C 180,E1 -12806.879,E2 -12806.879} C_VEL
LIN {X 0,Y 522.755,Z 340.657,A -85,B 0,C 180,E1 -12809.127,E2 -12809.127} C_VEL
LIN {X 0,Y 521.054,Z 333.138,A -85,B 0,C 180,E1 -12810.077,E2 -12810.077} C_VEL
LIN {X 0,Y 521.015,Z 333.145,A -85,B 0,C 180,E1 -12813.45,E2 -12813.45} C_VEL
LIN {X 0,Y 521.063,Z 333.132,A -85,B 0,C 180,E1 -12816.262,E2 -12816.262} C_VEL
LIN {X 0,Y 520.978,Z 333.151,A -85,B 0,C 180,E1 -12819.191,E2 -12819.191} C_VEL
LIN {X 0,Y 521.016,Z 333.138,A -85,B 0,C 180,E1 -12822.237,E2 -12822.237} C_VEL
LIN {X 0,Y 521.02,Z 333.14,A -85,B 0,C 180,E1 -12825.441,E2 -12825.441} C_VEL
LIN {X 0,Y 521.024,Z 333.146,A -85,B 0,C 180,E1 -12828.838,E2 -12828.838} C_VEL
LIN {X 0,Y 520.956,Z 333.148,A -85,B 0,C 180,E1 -12831.246,E2 -12831.246} C_VEL
LIN {X 0,Y 521.064,Z 333.132,A -85,B 0,C 180,E1 -12833.761,E2 -12833.761} C_VEL
LIN {X 0,Y 521.016,Z 333.147,A -85,B 0,C 180,E1 -12836.551,E2 -12836.551} C_VEL
LIN {X 0,Y 521,Z 333.141,A -85,B 0,C 180,E1 -12839.366,E2 -12839.366} C_VEL
LIN {X 0,Y 520.987,Z 333.144,A -85,B 0,C 180,E1 -12841.929,E2 -12841.929} C_VEL
LIN {X 0,Y 520.986,Z 333.148,A -85,B 0,C 180,E1 -12844.518,E2 -12844.518} C_VEL
LIN {X 0,Y 520.998,Z 333.141,A -85,B 0,C 180,E1 -12847.053,E2 -12847.053} C_VEL
LIN {X 0,Y 521.037,Z 333.137,A -85,B 0,C 180,E1 -12849.542,E2 -12849.542} C_VEL
LIN {X 0,Y 521.034,Z 333.137,A -85,B 0,C 180,E1 -12852.797,E2 -12852.797} C_VEL
LIN {X 0,Y 521.089,Z 333.137,A -85,B 0,C 180,E1 -12855.998,E2 -12855.998} C_VEL
LIN {X 0,Y 521.09,Z 333.131,A -85,B 0,C 180,E1 -12857.161,E2 -12857.161} C_VEL
LIN {X 0,Y 527.012,Z 350.374,A -85,B 0,C 180,E1 -12857.601,E2 -12857.601} C_VEL
LIN {X 0,Y 526.586,Z 393.24,A -85,B 0,C 180,E1 -12858.185,E2 -12858.185} C_VEL
LIN {X 0,Y 525.846,Z 399.083,A -85,B 0,C 180,E1 -12858.243,E2 -12858.243} C_VEL
LIN {X 0,Y 520.088,Z 418.055,A -85,B 0,C 180,E1 -12858.331,E2 -12858.331} C_VEL
LIN {X 0,Y 519.393,Z 423.895,A -85,B 0,C 180,E1 -12858.392,E2 -12858.392} C_VEL
LIN {X 0,Y 519.221,Z 456.196,A -85,B 0,C 180,E1 -12858.867,E2 -12858.867} C_VEL
LIN {X 0,Y 519.061,Z 470.33,A -85,B 0,C 180,E1 -12859.233,E2 -12859.233} C_VEL
LIN {X 0,Y 518.788,Z 483.953,A -85,B 0,C 180,E1 -12859.744,E2 -12859.744} C_VEL
LIN {X 0,Y 518.34,Z 496.679,A -85,B 0,C 180,E1 -12860.374,E2 -12860.374} C_VEL
LIN {X 0,Y 517.863,Z 507.68,A -85,B 0,C 180,E1 -12861.055,E2 -12861.055} C_VEL
LIN {X 0,Y 517.253,Z 520.309,A -85,B 0,C 180,E1 -12862.022,E2 -12862.022} C_VEL
LIN {X 0,Y 516.531,Z 530.687,A -85,B 0,C 180,E1 -12862.99,E2 -12862.99} C_VEL
LIN {X 0,Y 515.768,Z 540.992,A -85,B 0,C 180,E1 -12864.154,E2 -12864.154} C_VEL
LIN {X 0,Y 515.181,Z 549.489,A -85,B 0,C 180,E1 -12865.321,E2 -12865.321} C_VEL
LIN {X 0,Y 514.677,Z 557.641,A -85,B 0,C 180,E1 -12866.684,E2 -12866.684} C_VEL
LIN {X 0,Y 514.2,Z 564.212,A -85,B 0,C 180,E1 -12868.049,E2 -12868.049} C_VEL
LIN {X 0,Y 513.804,Z 568.742,A -85,B 0,C 180,E1 -12869.219,E2 -12869.219} C_VEL
LIN {X 0,Y 513.511,Z 573.435,A -85,B 0,C 180,E1 -12870.782,E2 -12870.782} C_VEL
LIN {X 0,Y 513.462,Z 576.67,A -85,B 0,C 180,E1 -12872.346,E2 -12872.346} C_VEL
LIN {X 0,Y 513.373,Z 578.569,A -85,B 0,C 180,E1 -12873.912,E2 -12873.912} C_VEL
LIN {X 0,Y 513.443,Z 579.157,A -85,B 0,C 180,E1 -12875.48,E2 -12875.48} C_VEL
LIN {X 0,Y 513.541,Z 578.459,A -85,B 0,C 180,E1 -12877.051,E2 -12877.051} C_VEL
LIN {X 0,Y 513.711,Z 576.453,A -85,B 0,C 180,E1 -12878.626,E2 -12878.626} C_VEL
LIN {X 0,Y 514.155,Z 573.058,A -85,B 0,C 180,E1 -12880.201,E2 -12880.201} C_VEL
LIN {X 0,Y 514.578,Z 568.193,A -85,B 0,C 180,E1 -12881.782,E2 -12881.782} C_VEL
LIN {X 0,Y 515.241,Z 561.683,A -85,B 0,C 180,E1 -12883.362,E2 -12883.362} C_VEL
LIN {X 0,Y 515.935,Z 554.39,A -85,B 0,C 180,E1 -12884.747,E2 -12884.747} C_VEL
LIN {X 0,Y 516.818,Z 545.273,A -85,B 0,C 180,E1 -12886.131,E2 -12886.131} C_VEL
LIN {X 0,Y 517.629,Z 535.71,A -85,B 0,C 180,E1 -12887.32,E2 -12887.32} C_VEL
LIN {X 0,Y 518.465,Z 525.055,A -85,B 0,C 180,E1 -12888.409,E2 -12888.409} C_VEL
LIN {X 0,Y 519.171,Z 514.278,A -85,B 0,C 180,E1 -12889.319,E2 -12889.319} C_VEL
LIN {X 0,Y 519.958,Z 501.512,A -85,B 0,C 180,E1 -12890.194,E2 -12890.194} C_VEL
LIN {X 0,Y 520.556,Z 488.675,A -85,B 0,C 180,E1 -12890.89,E2 -12890.89} C_VEL
LIN {X 0,Y 520.922,Z 475.727,A -85,B 0,C 180,E1 -12891.433,E2 -12891.433} C_VEL
LIN {X 0,Y 521.154,Z 461.603,A -85,B 0,C 180,E1 -12891.858,E2 -12891.858} C_VEL
LIN {X 0,Y 521.319,Z 447.214,A -85,B 0,C 180,E1 -12892.125,E2 -12892.125} C_VEL
LIN {X 0,Y 522.343,Z 354.837,A -85,B 0,C 180,E1 -12893.412,E2 -12893.412} C_VEL
LIN {X 0,Y 513.996,Z 334.357,A -85,B 0,C 180,E1 -12894.071,E2 -12894.071} C_VEL
LIN {X 0,Y 513.957,Z 334.027,A -85,B 0,C 180,E1 -12894.133,E2 -12894.133} C_VEL
LIN {X 0,Y 513.973,Z 334.026,A -85,B 0,C 180,E1 -12896.726,E2 -12896.726} C_VEL
LIN {X 0,Y 513.972,Z 334.02,A -85,B 0,C 180,E1 -12899.381,E2 -12899.381} C_VEL
LIN {X 0,Y 513.912,Z 334.03,A -85,B 0,C 180,E1 -12902.323,E2 -12902.323} C_VEL
LIN {X 0,Y 513.907,Z 334.026,A -85,B 0,C 180,E1 -12905.135,E2 -12905.135} C_VEL
LIN {X 0,Y 513.907,Z 334.029,A -85,B 0,C 180,E1 -12907.832,E2 -12907.832} C_VEL
LIN {X 0,Y 513.92,Z 334.026,A -85,B 0,C 180,E1 -12910.86,E2 -12910.86} C_VEL
LIN {X 0,Y 513.946,Z 334.027,A -85,B 0,C 180,E1 -12914.033,E2 -12914.033} C_VEL
LIN {X 0,Y 513.95,Z 334.02,A -85,B 0,C 180,E1 -12917.044,E2 -12917.044} C_VEL
LIN {X 0,Y 513.922,Z 334.025,A -85,B 0,C 180,E1 -12920.164,E2 -12920.164} C_VEL
LIN {X 0,Y 513.921,Z 334,A -85,B 0,C 180,E1 -12923.527,E2 -12923.527} C_VEL
LIN {X 0,Y 513.932,Z 334.023,A -85,B 0,C 180,E1 -12926.241,E2 -12926.241} C_VEL
LIN {X 0,Y 513.934,Z 334.016,A -85,B 0,C 180,E1 -12929.164,E2 -12929.164} C_VEL
LIN {X 0,Y 513.937,Z 334.023,A -85,B 0,C 180,E1 -12931.509,E2 -12931.509} C_VEL
LIN {X 0,Y 513.942,Z 334.017,A -85,B 0,C 180,E1 -12934.143,E2 -12934.143} C_VEL
LIN {X 0,Y 513.92,Z 334.023,A -85,B 0,C 180,E1 -12936.718,E2 -12936.718} C_VEL
LIN {X 0,Y 513.94,Z 334.018,A -85,B 0,C 180,E1 -12939.246,E2 -12939.246} C_VEL
LIN {X 0,Y 513.97,Z 334.029,A -85,B 0,C 180,E1 -12941.43,E2 -12941.43} C_VEL
LIN {X 0,Y 518.971,Z 350.82,A -85,B 0,C 180,E1 -12941.865,E2 -12941.865} C_VEL
LIN {X 0,Y 517.362,Z 453.791,A -85,B 0,C 180,E1 -12943.608,E2 -12943.608} C_VEL
LIN {X 0,Y 517.199,Z 469.252,A -85,B 0,C 180,E1 -12944.044,E2 -12944.044} C_VEL
LIN {X 0,Y 516.881,Z 482.769,A -85,B 0,C 180,E1 -12944.577,E2 -12944.577} C_VEL
LIN {X 0,Y 516.487,Z 496.254,A -85,B 0,C 180,E1 -12945.269,E2 -12945.269} C_VEL
LIN {X 0,Y 516.008,Z 509.879,A -85,B 0,C 180,E1 -12946.158,E2 -12946.158} C_VEL
LIN {X 0,Y 515.492,Z 522.133,A -85,B 0,C 180,E1 -12947.144,E2 -12947.144} C_VEL
LIN {X 0,Y 515.056,Z 533.175,A -85,B 0,C 180,E1 -12948.229,E2 -12948.229} C_VEL
LIN {X 0,Y 514.669,Z 543.09,A -85,B 0,C 180,E1 -12949.413,E2 -12949.413} C_VEL
LIN {X 0,Y 514.208,Z 551.331,A -85,B 0,C 180,E1 -12950.592,E2 -12950.592} C_VEL
LIN {X 0,Y 513.849,Z 559.219,A -85,B 0,C 180,E1 -12951.968,E2 -12951.968} C_VEL
LIN {X 0,Y 513.611,Z 565.541,A -85,B 0,C 180,E1 -12953.343,E2 -12953.343} C_VEL
LIN {X 0,Y 513.416,Z 570.837,A -85,B 0,C 180,E1 -12954.831,E2 -12954.831} C_VEL
LIN {X 0,Y 513.369,Z 574.179,A -85,B 0,C 180,E1 -12956.088,E2 -12956.088} C_VEL
LIN {X 0,Y 513.462,Z 575.754,A -85,B 0,C 180,E1 -12956.872,E2 -12956.872} C_VEL
LIN {X 0,Y 513.307,Z 577.84,A -85,B 0,C 180,E1 -12958.436,E2 -12958.436} C_VEL
LIN {X 0,Y 513.314,Z 578.525,A -85,B 0,C 180,E1 -12960,E2 -12960} C_VEL
LIN {X 0,Y 513.462,Z 577.799,A -85,B 0,C 180,E1 -12961.563,E2 -12961.563} C_VEL
LIN {X 0,Y 513.912,Z 575.633,A -85,B 0,C 180,E1 -12963.125,E2 -12963.125} C_VEL
LIN {X 0,Y 514.45,Z 571.94,A -85,B 0,C 180,E1 -12964.686,E2 -12964.686} C_VEL
LIN {X 0,Y 514.731,Z 566.723,A -85,B 0,C 180,E1 -12966.25,E2 -12966.25} C_VEL
LIN {X 0,Y 515.485,Z 560.747,A -85,B 0,C 180,E1 -12967.593,E2 -12967.593} C_VEL
LIN {X 0,Y 516.211,Z 553.065,A -85,B 0,C 180,E1 -12968.977,E2 -12968.977} C_VEL
LIN {X 0,Y 516.885,Z 545.059,A -85,B 0,C 180,E1 -12970.146,E2 -12970.146} C_VEL
LIN {X 0,Y 517.647,Z 535.347,A -85,B 0,C 180,E1 -12971.315,E2 -12971.315} C_VEL
LIN {X 0,Y 518.285,Z 525.671,A -85,B 0,C 180,E1 -12972.29,E2 -12972.29} C_VEL
LIN {X 0,Y 519.145,Z 513.923,A -85,B 0,C 180,E1 -12973.26,E2 -12973.26} C_VEL
LIN {X 0,Y 519.958,Z 501.152,A -85,B 0,C 180,E1 -12974.113,E2 -12974.113} C_VEL
LIN {X 0,Y 520.482,Z 486.919,A -85,B 0,C 180,E1 -12974.864,E2 -12974.864} C_VEL
LIN {X 0,Y 520.899,Z 472.912,A -85,B 0,C 180,E1 -12975.426,E2 -12975.426} C_VEL
LIN {X 0,Y 521.121,Z 458.172,A -85,B 0,C 180,E1 -12975.844,E2 -12975.844} C_VEL
LIN {X 0,Y 523.046,Z 385.13,A -85,B 0,C 180,E1 -12977.217,E2 -12977.217} C_VEL
LIN {X 0,Y 523.976,Z 355.798,A -85,B 0,C 180,E1 -12977.79,E2 -12977.79} C_VEL
LIN {X 0,Y 518.266,Z 343.18,A -85,B 0,C 180,E1 -12978.413,E2 -12978.413} C_VEL
LIN {X 0,Y 514.142,Z 334.894,A -85,B 0,C 180,E1 -12978.875,E2 -12978.875} C_VEL
LIN {X 0,Y 513.971,Z 334.023,A -85,B 0,C 180,E1 -12978.919,E2 -12978.919} C_VEL
LIN {X 0,Y 513.989,Z 334.021,A -85,B 0,C 180,E1 -12981.589,E2 -12981.589} C_VEL
LIN {X 0,Y 513.97,Z 334.026,A -85,B 0,C 180,E1 -12984.132,E2 -12984.132} C_VEL
LIN {X 0,Y 513.982,Z 334.02,A -85,B 0,C 180,E1 -12986.725,E2 -12986.725} C_VEL
LIN {X 0,Y 513.975,Z 334.02,A -85,B 0,C 180,E1 -12989.38,E2 -12989.38} C_VEL
LIN {X 0,Y 513.956,Z 334.02,A -85,B 0,C 180,E1 -12992.331,E2 -12992.331} C_VEL
LIN {X 0,Y 513.975,Z 334.016,A -85,B 0,C 180,E1 -12995.146,E2 -12995.146} C_VEL
